		rPlungeCycleGrindFeedGeometry:=1.0;
		IF (iAutoProcess = 1) AND xMicroRodActive THEN
			rPlungeCycleGrindFeedGeometry:=T_AutoGeometryPara.rPlungeCycleGrindFeedGeometry;
		END_IF;
		T_WorkTool.rToolRotationSpeed:=rToolRotationSpeed;
		xCalculation:=TRUE;
		WHILE(xCalculation) DO
			(* calculate the grinding way of each section *)
			FBCalcPlungeGrindingMultiCycle(	T_Geometry:= T_Geometry,
											T_AutoGeometryPara:= T_AutoGeometryPara,
											rToolDiameter:= rToolDiameter,
											rToolDiameterWithOffset:=rToolDiameterWithOffset,
											rPlungeCycleGrindFeedGeometry:=rPlungeCycleGrindFeedGeometry,
											iStartSection:= iStartSection,
											iEndSection:= iEndSection,
											xReset:= xResetFB,
											xInit:=xInitFB);
			IF FBCalcPlungeGrindingMultiCycle.xEndWorking THEN		(* check if the end of the to work Tool is reached *)
				xCalculation:=FALSE;
				EXIT;
			END_IF;
			IF (FBCalcPlungeGrindingMultiCycle.iStepSectionWork = 7) THEN
				(* Count the Plunge Cycle *)
				T_WorkTool.iTotalCountDownPlungeCycle:=T_WorkTool.iTotalCountDownPlungeCycle + 1;
			END_IF;
			IF (FBCalcPlungeGrindingMultiCycle.iStepSectionWork >= 1) AND (FBCalcPlungeGrindingMultiCycle.iStepSectionWork <= 6) THEN
			(* section 1 - 6 *)
				iTmpStartSection:=iStartSection + (FBCalcPlungeGrindingMultiCycle.iStepSectionWork - 1);
				rGrindFeederPlunge:=FBCalcPlungeGrindingMultiCycle.rGrindingRelativePosition;
				T_WorkTool.rGrindFeederPlunge:=rGrindFeederPlunge;
				T_WorkTool.rPitch:=T_Geometry.arSectionPitch[iTmpStartSection];
				T_WorkTool.rToolLength:=T_Geometry.arSectionLength[iTmpStartSection];
				FBToolCalcul(	xMicroRodActive:=xMicroRodActive,
								xBeckhoffDriveActive:=FALSE,
								T_WorkTool:= T_WorkTool);
				rTimeLeftWork:=rTimeLeftWork + T_WorkTool.rTimeLeftWork;
			END_IF;
			IF (FBCalcPlungeGrindingMultiCycle.iStepSectionWork = 0) THEN
				(* Calc Plunge *)
				IF T_AutoGeometryPara.xPlungeActivationGeometry THEN
					T_WorkTool.rPitch:=T_Geometry.arSectionPitch[iStartSection] * -1.0;
					T_WorkTool.rGrindFeederPlunge:=FBCalcPlungeGrindingMultiCycle.rGrindingRelativePosition;
					rToolFeedLength:=T_AutoGeometryPara.rPlungeLengthToolFeedGeometry;
					T_WorkTool.rToolLength:=rToolFeedLength;
					T_WorkTool.rToolRotationSpeed:=T_AutoGeometryPara.rSpeedToolRotationGeometry;
					FBToolCalcul(	xMicroRodActive:=xMicroRodActive,
									xBeckhoffDriveActive:=FALSE,
									T_WorkTool:= T_WorkTool);
					rSpeedToolFeed:=T_WorkTool.rToolFeederSpeedUnit * -1.0;
					IF (rSpeedToolFeed <> 0) THEN
						rTimeLeftWork:=rTimeLeftWork + T_WorkTool.rToolLength/rSpeedToolFeed;
					END_IF;
				ELSE
					(* No Plunging activation, than also is the GrindFeeder the master *)
					rPlungeGrind:=ABS(FBCalcPlungeGrindingMultiCycle.rGrindingRelativePosition);
					IF (T_AutoGeometryPara.rPlungeSpeedGrindFeedGeometry <> 0) THEN
						rTimeLeftWork:=rTimeLeftWork + (rPlungeGrind / T_AutoGeometryPara.rPlungeSpeedGrindFeedGeometry);
					END_IF;
				END_IF;
			END_IF;
			IF (FBCalcPlungeGrindingMultiCycle.iStepSectionWork = 7) THEN
				(* Calc Displace *)
				IF T_AutoGeometryPara.xDisplaceActivationGeometry THEN
					T_WorkTool.rPitch:=T_Geometry.arSectionPitch[iEndSection] * -1.0;
					T_WorkTool.rGrindFeederPlunge:=FBCalcPlungeGrindingMultiCycle.rGrindingRelativePosition;
					rToolFeedLength:=T_AutoGeometryPara.rDisplaceLengthToolFeedGeometry;
					T_WorkTool.rToolLength:=rToolFeedLength;
					T_WorkTool.rToolRotationSpeed:=T_AutoGeometryPara.rSpeedToolRotationGeometry;
					FBToolCalcul(	xMicroRodActive:=xMicroRodActive,
									xBeckhoffDriveActive:=FALSE,
									T_WorkTool:= T_WorkTool);
					rSpeedToolFeed:=T_WorkTool.rToolFeederSpeedUnit * -1.0;
					IF (rSpeedToolFeed <> 0) THEN
						rTimeLeftWork:=rTimeLeftWork + T_WorkTool.rToolLength/rSpeedToolFeed;
					END_IF;
				ELSE
					(* No Displace activation, than also is the GrindFeeder the master *)
					rDisplaceGrind:=ABS(FBCalcPlungeGrindingMultiCycle.rGrindingRelativePosition);
					IF (T_AutoGeometryPara.rDisplaceSpeedGrindFeedGeometry <> 0) THEN
						rTimeLeftWork:=rTimeLeftWork + (rDisplaceGrind / T_AutoGeometryPara.rDisplaceSpeedGrindFeedGeometry);
					END_IF;
				END_IF;
			END_IF;
		END_WHILE;
		IF (T_AutoGeometryPara.iCycleGeometry > 1) THEN
			rTimeLeftWork:=rTimeLeftWork * INT_TO_REAL(T_AutoGeometryPara.iCycleGeometry);
		END_IF;
	END_IF;
(**************iAutoProcess 2 --> AutoGroove********************************************************************************************************************************************************************************************************)
	IF (iAutoProcess = 2) THEN
	(* calculate the time for the process AutoGeometry or AutoGroove *)
		T_WorkTool.iTotalCountDownPlungeCycle:=0;
		(* Check Start and End Section of the ToolGeometry *)
		FOR ii:=1 TO 6 DO
			IF T_Geometry.axActiveSection[ii] THEN
				IF (iStartSection = 0) THEN
					iStartSection:=ii;
				END_IF;
				iEndSection:=ii;
			END_IF;
		END_FOR;
(*
		xResetFB:=TRUE;
		(* reset first the FB for calculate the grinding plunge for each sections *)
		FBCalcPlungeGrinding(	rToolDiameter:= rToolDiameter,
								rToolDiameterWithOffset:=rToolDiameterWithOffset,
								xReset:= xResetFB);
		rPlungeCycleGrindFeedGeometry:=1.0;
*)
		xResetFB:=TRUE;
		(* reset first the FB for calculate the grinding plunge for each sections *)
		FBCalcPlungeGrindingMultiCycle(	rToolDiameter:= rToolDiameter,
										rToolDiameterWithOffset:=rToolDiameterWithOffset,
										xReset:= xResetFB,
										xInit:=xInitFB);
		xInitFB:=TRUE;
		FBCalcPlungeGrindingMultiCycle(	T_Geometry:= T_Geometry,
										T_AutoGeometryPara:= T_AutoGeometryPara,
										rToolDiameter:= rToolDiameter,
										rToolDiameterWithOffset:=rToolDiameterWithOffset,
										rPlungeCycleGrindFeedGeometry:=rPlungeCycleGrindFeedGeometry,
										iStartSection:= iStartSection,
										iEndSection:= iEndSection,
										xReset:= xResetFB,
										xInit:=xInitFB);
		rPlungeCycleGrindFeedGeometry:=1.0;
		IF (iAutoProcess = 2) OR NOT(xMicroRodActive) THEN
			rPlungeCycleGrindFeedGeometry:=rToolDiameter;		(* for the groove process or for the MicroWire is not possible to work in more cycle, because of that it will set the tooldiamter *)
		END_IF;
		T_WorkTool.rToolRotationSpeed:=rToolRotationSpeed;
		xCalculation:=TRUE;
		WHILE(xCalculation) DO
			(* calculate the grinding way of each section *)
			FBCalcPlungeGrindingMultiCycle(	T_Geometry:= T_Geometry,
											T_AutoGeometryPara:= T_AutoGeometryPara,
											rToolDiameter:= rToolDiameter,
											rToolDiameterWithOffset:=rToolDiameterWithOffset,
											rPlungeCycleGrindFeedGeometry:=rPlungeCycleGrindFeedGeometry,
											iStartSection:= iStartSection,
											iEndSection:= iEndSection,
											xReset:= xResetFB,
											xInit:=xInitFB);
			IF FBCalcPlungeGrindingMultiCycle.xEndWorking THEN		(* check if the end of the to work Tool is reached *)
				xCalculation:=FALSE;
				EXIT;
			END_IF;
			IF (T_WorkTool.iTotalCountDownPlungeCycle >= 20) THEN	(* not possible to work a Tool in more that 20 cycle *)
				xCalculation:=FALSE;
				EXIT;
			END_IF;
			IF (FBCalcPlungeGrindingMultiCycle.iStepSectionWork = 7) THEN
				(* Count the Plunge Cycle *)
				T_WorkTool.iTotalCountDownPlungeCycle:=T_WorkTool.iTotalCountDownPlungeCycle + 1;
			END_IF;
			IF (FBCalcPlungeGrindingMultiCycle.iStepSectionWork >= 1) AND (FBCalcPlungeGrindingMultiCycle.iStepSectionWork <= 6) THEN
			(* section 1 - 6 *)
				iTmpStartSection:=iStartSection + (FBCalcPlungeGrindingMultiCycle.iStepSectionWork - 1);
				rGrindFeederPlunge:=FBCalcPlungeGrindingMultiCycle.rGrindingRelativePosition;
				T_WorkTool.rGrindFeederPlunge:=rGrindFeederPlunge;
				T_WorkTool.rPitch:=T_AutoGroovePara.rPitchGroove;
				T_WorkTool.rToolLength:=T_Geometry.arSectionLength[iTmpStartSection];
				FBToolCalcul(	xMicroRodActive:=xMicroRodActive,
								xBeckhoffDriveActive:=FALSE,
								T_WorkTool:= T_WorkTool);
				rTimeLeftWork:=rTimeLeftWork + T_WorkTool.rTimeLeftWork;
			END_IF;
			IF (FBCalcPlungeGrindingMultiCycle.iStepSectionWork = 0) THEN
				(* Calc Plunge *)
				IF T_AutoGroovePara.xPlungeActivationGroove  THEN
					T_WorkTool.rPitch:=T_AutoGroovePara.rPitchGroove * -1.0;
					T_WorkTool.rGrindFeederPlunge:=FBCalcPlungeGrindingMultiCycle.rGrindingRelativePosition;
					rToolFeedLength:=T_AutoGroovePara.rPlungeLengthToolFeedGroove;
					T_WorkTool.rToolLength:=rToolFeedLength;
					T_WorkTool.rToolRotationSpeed:=T_AutoGroovePara.rSpeedToolRotationGroove;
					FBToolCalcul(	xMicroRodActive:=xMicroRodActive,
									xBeckhoffDriveActive:=FALSE,
									T_WorkTool:= T_WorkTool);
					rSpeedToolFeed:=T_WorkTool.rToolFeederSpeedUnit * -1.0;
					IF (rSpeedToolFeed <> 0) THEN
						rTimeLeftWork:=rTimeLeftWork + T_WorkTool.rToolLength/rSpeedToolFeed;
					END_IF;
				ELSE
					(* No Plunging activation, than also is the GrindFeeder the master *)
					rPlungeGrind:=ABS(FBCalcPlungeGrindingMultiCycle.rGrindingRelativePosition);
					IF (T_AutoGroovePara.rPlungeSpeedGrindFeedGroove <> 0) THEN
						rTimeLeftWork:=rTimeLeftWork + (rPlungeGrind / T_AutoGroovePara.rPlungeSpeedGrindFeedGroove);
					END_IF;
				END_IF;
			END_IF;
			IF (FBCalcPlungeGrindingMultiCycle.iStepSectionWork = 7) THEN
				(* Calc Displace *)
				IF T_AutoGroovePara.xDisplaceActivationGroove  THEN
					T_WorkTool.rPitch:=T_AutoGroovePara.rPitchGroove * -1.0;
					T_WorkTool.rGrindFeederPlunge:=FBCalcPlungeGrindingMultiCycle.rGrindingRelativePosition;
					rToolFeedLength:=T_AutoGroovePara.rDisplaceLengthToolFeedGroove;
					T_WorkTool.rToolLength:=rToolFeedLength;
					T_WorkTool.rToolRotationSpeed:=T_AutoGroovePara.rSpeedToolRotationGroove;
					FBToolCalcul(	xMicroRodActive:=xMicroRodActive,
									xBeckhoffDriveActive:=FALSE,
									T_WorkTool:= T_WorkTool);
					rSpeedToolFeed:=T_WorkTool.rToolFeederSpeedUnit * -1.0;
					IF (rSpeedToolFeed <> 0) THEN
						rTimeLeftWork:=rTimeLeftWork + T_WorkTool.rToolLength/rSpeedToolFeed;
					END_IF;
				ELSE
					(* No Displace activation, than also is the GrindFeeder the master *)
					rDisplaceGrind:=ABS(FBCalcPlungeGrindingMultiCycle.rGrindingRelativePosition);
					IF (T_AutoGroovePara.rDisplaceSpeedGrindFeedGroove <> 0) THEN
						rTimeLeftWork:=rTimeLeftWork + (rPlungeGrind / T_AutoGroovePara.rDisplaceSpeedGrindFeedGroove);
					END_IF;
				END_IF;
			END_IF;
		END_WHILE;
		IF (T_AutoGroovePara.iNumberOfGrooves > 1) THEN
			rTimeLeftWork:=rTimeLeftWork * INT_TO_REAL(T_AutoGroovePara.iNumberOfGrooves);
			(* Berechnung zusätzlicher Weg und Zeit für Ausstechen & Einstechen ab 2. Zyklus*)
			rPlungeGrind:=ABS(T_ProcessPara.rSecurityPosGrindFeedProcess - T_ProcessPara.rToolDiameterProcess) * 2.0;
			rTimeAddLeftWorkPlungeGrind:= rPlungeGrind / T_ProcessPara.rSpeedForwardFastGrindFeed;
			(* Berechnung zusätzlicher Weg und Zeit  Ausstechen für letzten Zyklus*)
			rPlungeGrind2:=ABS(T_ProcessPara.rSecurityPosGrindFeedProcess - T_ProcessPara.rToolDiameterProcess);
			rTimeAddLeftWorkPlungeGrind2:= rPlungeGrind2 / T_ProcessPara.rSpeedForwardFastGrindFeed;
			(*Berechnung zusätzlicher Weg und Zeit  Rückfahren  ab 2. Zyklus*)
			rToolLength:=0;
			FOR ii:=1 TO 6 DO
				IF T_Geometry.axActiveSection[ii] THEN
					rToolLength:=rToolLength + T_Geometry.arSectionLength[ii];
				END_IF;
			END_FOR;
			rTimeAddLeftWorkToolFeed:= rToolLength*10/T_ProcessPara.rSpeedStartPosToolFeedProcess;
			(*Berchnung der gesamten zusätzlichen Prozesszeit*)
			rTimeAddLeftWork:=(rTimeAddLeftWorkPlungeGrind + rTimeAddLeftWorkToolFeed) * (T_AutoGroovePara.iNumberOfGrooves -1);
			rTimeAddLeftWork:= rTimeAddLeftWork+rTimeAddLeftWorkPlungeGrind2;
			rTimeLeftWork:=rTimeLeftWork + rTimeAddLeftWork;
		END_IF;
	END_IF;
(**************iAutoProcess 0***********************************************************************************************************************************************************************************************************************)
	IF (iAutoProcess = 0) THEN
	(* Calculate the time for the process ToolCalibration *)
		T_WorkTool.rToolRotationSpeed:=T_CalibrationPara.rSpeedToolRotationCalib;
		T_WorkTool.rGrindFeederPlunge:=T_ProcessPara.rOffsetBeforeToolDiaGrindFeedProcess;
		T_WorkTool.rPitch:=T_CalibrationPara.rPitchCalib;
		T_WorkTool.rToolLength:=T_CalibrationPara.rToolLengthCylinderPartCalib;
		FBToolCalcul(	xMicroRodActive:=xMicroRodActive,
						xBeckhoffDriveActive:=FALSE,
						T_WorkTool:= T_WorkTool);
		rTimeLeftWork:=rTimeLeftWork + T_WorkTool.rTimeLeftWork;
		IF T_CalibrationPara.xPlungeActivationCalib THEN
			T_WorkTool.rPitch:=T_CalibrationPara.rPitchCalib;
			T_WorkTool.rGrindFeederPlunge:=T_ProcessPara.rOffsetBeforeToolDiaGrindFeedProcess;
			rToolFeedLength:=T_CalibrationPara.rPlungeLengthToolFeedCalib;
			T_WorkTool.rToolLength:=rToolFeedLength;
			FBToolCalcul(	xMicroRodActive:=xMicroRodActive,
							xBeckhoffDriveActive:=FALSE,
							T_WorkTool:= T_WorkTool);
			rSpeedToolFeed:=T_WorkTool.rToolFeederSpeedUnit;
			IF (rSpeedToolFeed <> 0) THEN
				rTimeLeftWork:=rTimeLeftWork + T_WorkTool.rToolLength/ABS(rSpeedToolFeed);
			END_IF;
		ELSE
			(* No Plunging activation, than also is the GrindFeeder the master *)
			rPlungeGrind:=T_ProcessPara.rOffsetBeforeToolDiaGrindFeedProcess;
			rTimeLeftWork:=rTimeLeftWork + (rPlungeGrind / T_CalibrationPara.rPlungeSpeedGrindFeedCalib);
		END_IF;


		IF T_CalibrationPara.xDisplaceActivationCalib THEN
			T_WorkTool.rPitch:=T_CalibrationPara.rPitchCalib * -1.0;
			T_WorkTool.rGrindFeederPlunge:=T_ProcessPara.rOffsetBeforeToolDiaGrindFeedProcess;
			rToolFeedLength:=T_CalibrationPara.rDisplaceLengthToolFeedCalib;
			T_WorkTool.rToolLength:=rToolFeedLength;
			FBToolCalcul(	xMicroRodActive:=xMicroRodActive,
							xBeckhoffDriveActive:=FALSE,
							T_WorkTool:= T_WorkTool);
			rSpeedToolFeed:=T_WorkTool.rToolFeederSpeedUnit;
			IF (rSpeedToolFeed <> 0) THEN
				rTimeLeftWork:=rTimeLeftWork + T_WorkTool.rToolLength/ABS(rSpeedToolFeed);
			END_IF;
		ELSE
			(* No Displace activation, than also is the GrindFeeder the master *)
			rDisplaceGrind:=T_ProcessPara.rOffsetBeforeToolDiaGrindFeedProcess;
			rTimeLeftWork:=rTimeLeftWork + (rDisplaceGrind / T_CalibrationPara.rDisplaceSpeedGrindFeedCalib);
		END_IF;
	END_IF;
	rProcessTime:=rTimeLeftWork;
END_FUNCTION_BLOCK

(* POU GENERAL/FB_TOOL_CALCUL, ST *)
FUNCTION_BLOCK FB_TOOL_CALCUL
VAR_INPUT
	xMicroRodActive: BOOL;			(* choice of the machine MicroWire or MicroRod *)
	xBeckhoffDriveActive: BOOL;		(* choice of the Axis Beckhoff or EcoStep *)
END_VAR
VAR_IN_OUT
	T_WorkTool:ST_WORKTOOL;		(* Tool Parameter *)
END_VAR
VAR_OUTPUT
END_VAR
VAR
END_VAR
(****************************************************************************************************************************************************)
(***********                                  This Functionblock calculate all needed parameter for work a Tool                                            ************)
(****************************************************************************************************************************************************)
(* calcul ToolRotation Speed in inc/64s *)
	IF (T_WorkTool.rToolRotationSpeed <> 0) AND (T_WorkTool.rToolRightGearRatio <> 0) THEN
		T_WorkTool.rToolRotationSpeedMotor:=((T_WorkTool.rToolRotationSpeed / 60.0) * 8000.0 * 64.0) / T_WorkTool.rToolRightGearRatio;
	ELSE
		RETURN;	(* Exit FB *)
	END_IF;
(* calcul ToolFeeder Speed in mm/s *)
	T_WorkTool.rToolFeederSpeedUnit:=T_WorkTool.rPitch * (T_WorkTool.rToolRotationSpeed / 60.0);
(* calcul ToolFeeder Speed in inc/64s Relativ *)
	T_WorkTool.rToolFeederSpeedMotorRel:=T_WorkTool.rToolFeederScaleFactor * T_WorkTool.rToolFeederSpeedUnit * 64.0;
(* calcul ToolFeeder Speed in inc/64s Relativ *)
	T_WorkTool.rToolFeederSpeedMotorAbs:=(T_WorkTool.rToolRotationSpeedMotor * T_WorkTool.rToolRightGearRatio) + T_WorkTool.rToolFeederSpeedMotorRel;
(* Set ToolFeeder GearDivider *)
	T_WorkTool.iToolFeederGearDivider:=T_WorkTool.iBaseGearDivider;
	IF xMicroRodActive THEN
	(* calcul ToolFeeder GearFactor *)
		IF (T_WorkTool.rPitch <> 0) THEN
			T_WorkTool.iToolFeederGearFactor:=REAL_TO_INT(INT_TO_REAL(T_WorkTool.iBaseGearDivider) / (T_WorkTool.rToolRotationSpeedMotor / T_WorkTool.rToolFeederSpeedMotorRel));
		ELSE
			T_WorkTool.iToolFeederGearFactor:=REAL_TO_INT(INT_TO_REAL(T_WorkTool.iToolFeederGearDivider) * T_WorkTool.rToolRightGearRatio);
		END_IF;
	ELSE
	(* calcul ToolFeeder GearFactor *)
		IF (T_WorkTool.rPitch <> 0) THEN
			T_WorkTool.iToolFeederGearFactor:=REAL_TO_INT(INT_TO_REAL(T_WorkTool.iBaseGearDivider) / (T_WorkTool.rToolRotationSpeedMotor / T_WorkTool.rToolFeederSpeedMotorAbs));
		ELSE
			T_WorkTool.iToolFeederGearFactor:=REAL_TO_INT(INT_TO_REAL(T_WorkTool.iToolFeederGearDivider) * T_WorkTool.rToolRightGearRatio);
		END_IF;
	END_IF;
(* calcul Time to work *)
	IF (T_WorkTool.rToolFeederSpeedUnit <> 0) THEN
		T_WorkTool.rTimeLeftWork:=(T_WorkTool.rToolLength * 10.0) / ABS(T_WorkTool.rToolFeederSpeedUnit);
	ELSE
		T_WorkTool.rTimeLeftWork:=0.0;
	END_IF;
(* calcul ToolFeeder relative Position to drive *)
	T_WorkTool.rToolFeederRelPositionUnit:=T_WorkTool.rToolLength * 10.0;
	T_WorkTool.rToolFeederRelPositionMotor:=T_WorkTool.rToolFeederRelPositionUnit * T_WorkTool.rToolFeederScaleFactor;
(* calcul GrindFeeder Speed in um/s *)
	IF (T_WorkTool.rTimeLeftWork <> 0) THEN
		T_WorkTool.rGrindFeederSpeedUnit:=T_WorkTool.rGrindFeederPlunge / T_WorkTool.rTimeLeftWork;
	ELSE
		T_WorkTool.rGrindFeederSpeedUnit:=0.0;
	END_IF;
(* calcul GrindFeeder Speed in inc/s *)
	T_WorkTool.rGrindFeederSpeedMotor:=T_WorkTool.rGrindFeederSpeedUnit * T_WorkTool.rGrindFeederScaleFactor * 64.0;
END_FUNCTION_BLOCK

(* POU GENERAL/FB_CALC_PLUNGE_GRINDING, ST *)
FUNCTION_BLOCK FB_CALC_PLUNGE_GRINDING
VAR_INPUT
	T_Geometry:ST_GEOMETRY;								(* Structure of the NovRAM parameter *)
	T_AutoGeometryPara:ST_EXCHG_PARAM_AUTOGEOMETRY;	(* Structure of the NovRAM parameter *)
	rToolDiameter:REAL;					(* diameter of the unworked Tool *)
	rToolDiameterWithOffset:REAL;			(* diameter of the unworked Tool plus the offset for plunge and displace procedure *)
	rPlungeCycleGrindFeedGeometry:REAL;	(* max grinding plunging per cycle *)
	iStartSection:INT;						(* number of the start section *)
	iEndSection:INT;						(* number of the end section *)
END_VAR
VAR_IN_OUT
	xReset:BOOL;						(* resetting of the FB *)
END_VAR
VAR_OUTPUT
	iStepSectionWork:INT;				(* actual worked section number *)
	rGrindingRelativePosition:REAL;		(* relative way of the GrindFeeder plunge *)
	xEndWorking:BOOL;				(* end of the hole working procedure *)
	xError:BOOL;						(* error flag *)
END_VAR
VAR
(***S***)
	rActualPositionGrindFeedStart: ARRAY [0..7] OF REAL;	(* 0=StartPos Plunge,1-6=Dynamic StartPos Section 1-6, 7=StartPos Displace *)
	rActualPositionGrindFeedEnd: ARRAY [0..7] OF REAL;	(* 0=EndPos Plunge,1-6=Dynamic EndPos Section 1-6, 7=EndPos Displace *)
	rDistanceToWorkedTool: REAL;
	ii: INT;
	iStepSection: INT;
	axWorkEndSection: ARRAY [0..7] OF BOOL;
	xCheckEnd: BOOL;
	rTmpActualPositionGrindFeedStart:REAL;
	iStepCheckSection: INT;
	rTmpDistance: REAL;
	rGrinded: REAL;
END_VAR
(****************************************************************************************************************************************************)
(***********      This Functionblock calculate the plunge way for the GrindFeeder axis for the geometry sections  1-6        ************)
(***********                                           It calculate also the plunge and displace procedure							    ************)
(****************************************************************************************************************************************************)
IF xReset THEN
	xReset:=FALSE;
	iStepSection:=0;
	FOR ii:=0 TO 7 DO
		rActualPositionGrindFeedStart[ii]:=rToolDiameterWithOffset;
		rActualPositionGrindFeedEnd[ii]:=rToolDiameterWithOffset;
		axWorkEndSection[ii]:=FALSE;
	END_FOR;
	rActualPositionGrindFeedStart[0]:=rToolDiameterWithOffset;
	rActualPositionGrindFeedEnd[7]:=rToolDiameterWithOffset;
	rTmpActualPositionGrindFeedStart:=rToolDiameterWithOffset;
	rGrindingRelativePosition:=0.0;
	iStepSectionWork:=0;
	RETURN;
END_IF;
xError:=FALSE;
(* check the settled start and end section *)
IF (iStartSection < 1) OR (iStartSection > 6) THEN
	xError:=TRUE;
	RETURN;
END_IF;
IF (iEndSection < 1) OR (iEndSection > 6) THEN
	xError:=TRUE;
	RETURN;
END_IF;
IF (iStepSection < 0) OR (iStepSection > 7) THEN
	xError:=TRUE;
	RETURN;
END_IF;

CASE iStepSection OF
	(* plunge procedure *)
		0:	iStepCheckSection:=1;
			xCheckEnd:=TRUE;
			(* Check if the end of all section is reached *)
			FOR ii:=iStartSection TO iEndSection DO
				IF (rActualPositionGrindFeedStart[iStepCheckSection] <> T_Geometry.arStartDiameter[ii]) THEN
					xCheckEnd:=FALSE;
				END_IF;
				IF (rActualPositionGrindFeedEnd[iStepCheckSection] <> T_Geometry.arEndDiameter[ii]) THEN
					xCheckEnd:=FALSE;
				END_IF;
				iStepCheckSection:=iStepCheckSection + 1;
			END_FOR;
			xEndWorking:=xCheckEnd;
			IF xEndWorking THEN
				rGrindingRelativePosition:=0.0;
				RETURN;
			END_IF;
			IF (T_Geometry.arStartDiameter[iStartSection] = rActualPositionGrindFeedEnd[0]) THEN	(* check if the defined ToolDiameter for the plunge procedure is reached *)
				axWorkEndSection[0]:=TRUE;
				rGrindingRelativePosition:=rToolDiameterWithOffset - T_Geometry.arStartDiameter[iStartSection];
			END_IF;
			IF NOT(axWorkEndSection[0]) THEN
			(* if the end of the plunge procedure is not reached, then calculate the plunge way of the plunge procedure *)
				rGrindingRelativePosition:=(rToolDiameterWithOffset - rActualPositionGrindFeedEnd[0]) + rPlungeCycleGrindFeedGeometry;
				IF ((rToolDiameterWithOffset - rGrindingRelativePosition) <= T_Geometry.arStartDiameter[iStartSection]) THEN
					rGrindingRelativePosition:=rToolDiameterWithOffset - T_Geometry.arStartDiameter[iStartSection];
				END_IF;
			END_IF;
			rActualPositionGrindFeedStart[0]:=rToolDiameterWithOffset;	(* the start zero section of the geometry is always the diameter of the Tool *)
			rActualPositionGrindFeedEnd[0]:=rToolDiameterWithOffset - rGrindingRelativePosition;	(* calcualte the plunge way *)
			iStepSectionWork:=iStepSection;	(* set the actual section which is working *)
			iStepSection:=iStepSection + 1;		(* go to the next section *)
	(* geometry section 1,2,3,4,5 and 6 *)
	1,2,3,4,5,6:	rGrinded:=(rActualPositionGrindFeedStart[iStepSection] - rActualPositionGrindFeedEnd[iStepSection - 1]);	(* calculate the difference of the worked section before to the unworked section after *)
			IF (rGrinded < 0) THEN
				rGrinded:=rGrinded;
			END_IF;
			rActualPositionGrindFeedStart[iStepSection]:=rActualPositionGrindFeedStart[iStepSection] - rGrinded;		(* set the new diameter of the section which will go to work *)
			rTmpDistance:=T_Geometry.arStartDiameter[iStartSection + (iStepSection - 1)] - T_Geometry.arEndDiameter[iStartSection + (iStepSection - 1)]; (* set the difference of the start and end diameter of the section *)
			IF (rActualPositionGrindFeedStart[iStepSection] < T_Geometry.arStartDiameter[iStartSection + (iStepSection - 1)]) THEN	(* correct of the to grind Tool diameter *)
				rActualPositionGrindFeedStart[iStepSection]:=T_Geometry.arStartDiameter[iStartSection + (iStepSection - 1)];
			END_IF;
			rGrindingRelativePosition:=rPlungeCycleGrindFeedGeometry - rGrinded;	(* calculate the effectiv way for the plunge *)
			IF (rGrinded >= rPlungeCycleGrindFeedGeometry) THEN				(* check if the to grinding way is grater than the defined max grinding *)
				IF (rActualPositionGrindFeedStart[iStepSection] < T_Geometry.arEndDiameter[iStartSection + (iStepSection - 1)]) THEN
				(* correct the effective way for the plunge, because it can not work more than the defined grinding way *)
					rGrindingRelativePosition:=rActualPositionGrindFeedStart[iStepSection] - T_Geometry.arEndDiameter[iStartSection + (iStepSection - 1)];
				END_IF;
			ELSE
				IF (rTmpDistance = 0) THEN
				(* a cylinder part will now work *)
					rGrindingRelativePosition:=0.0;
				ELSE
					(* a cone part will now work *)
					rTmpDistance:=T_Geometry.arStartDiameter[iStartSection + (iStepSection - 1)] - rActualPositionGrindFeedEnd[iStepSection];
					rGrindingRelativePosition:=rTmpDistance + rPlungeCycleGrindFeedGeometry;
					IF ((T_Geometry.arStartDiameter[iStartSection + (iStepSection - 1)] - rGrindingRelativePosition) < T_Geometry.arEndDiameter[iStartSection + (iStepSection - 1)]) THEN
					(* correct the effective way for the plunge, because it can not work more than the defined grinding way *)
						rGrindingRelativePosition:=T_Geometry.arStartDiameter[iStartSection + (iStepSection - 1)] - T_Geometry.arEndDiameter[iStartSection + (iStepSection - 1)];
					END_IF;
				END_IF;
			END_IF;
			rActualPositionGrindFeedEnd[iStepSection]:=rActualPositionGrindFeedStart[iStepSection] - rGrindingRelativePosition;	(* calculate the end position of the section *)
			iStepSectionWork:=iStepSection;		(* set the actual section which is working *)
			IF ((iStepSection + (iStartSection - 1)) < iEndSection) THEN	(* check if the end section is active *)
				iStepSection:=iStepSection + 1;
			ELSE
				iStepSection:=7;	(* end section is reached-->go the displace procedure *)
			END_IF;
	(* plunge procedure *)
	7:		rActualPositionGrindFeedStart[7]:=rActualPositionGrindFeedEnd[iEndSection - (iStartSection - 1)];	(* set the new diameter of the section which will going to work *)
			rDistanceToWorkedTool:=rActualPositionGrindFeedStart[7] - rToolDiameterWithOffset;	(* check the distance to the end diameter, which will go to work *)
			rGrindingRelativePosition:=rDistanceToWorkedTool;
			IF (rActualPositionGrindFeedStart[5] = T_Geometry.arEndDiameter[iEndSection]) THEN
				axWorkEndSection[7]:=TRUE;		(* the end of this section is reached *)
			ELSE
				axWorkEndSection[7]:=FALSE;		(* the end of this section is reached *)
			END_IF;
			rActualPositionGrindFeedEnd[7]:=rToolDiameterWithOffset;
			iStepSectionWork:=iStepSection;		(* set the actual section which is working *)
			iStepSection:=0;
END_CASE;
END_FUNCTION_BLOCK

(* POU GENERAL/FB_CALC_PLUNGE_GRINDING_MultiCycle, ST *)
FUNCTION_BLOCK FB_CALC_PLUNGE_GRINDING_MultiCycle
VAR_INPUT
	T_Geometry:ST_GEOMETRY;								(* Structure of the NovRAM parameter *)
	T_AutoGeometryPara:ST_EXCHG_PARAM_AUTOGEOMETRY;	(* Structure of the NovRAM parameter *)
	rToolDiameter:REAL;					(* diameter of the unworked Tool *)
	rToolDiameterWithOffset:REAL;			(* diameter of the unworked Tool plus the offset for plunge and displace procedure *)
	rPlungeCycleGrindFeedGeometry:REAL;	(* max grinding plunging per cycle *)
	iStartSection:INT;						(* number of the start section *)
	iEndSection:INT;						(* number of the end section *)
END_VAR
VAR_IN_OUT
	xReset:BOOL;						(* resetting of the FB *)
	xInit:BOOL;							(* Init of the FB *)
END_VAR
VAR_OUTPUT
	iStepSectionWork:INT;				(* actual worked section number *)
	rGrindingRelativePosition:REAL;		(* relative way of the GrindFeeder plunge *)
	xEndWorking:BOOL;				(* end of the hole working procedure *)
	xError:BOOL;						(* error flag *)
END_VAR
VAR
	rActualPositionGrindFeedStart: ARRAY [0..7] OF REAL;	(* 0=StartPos Plunge,1-4=Dynamic StartPos Section 1-4, 5=StartPos Displace *)
	rActualPositionGrindFeedEnd: ARRAY [0..7] OF REAL;	(* 0=EndPos Plunge,1-4=Dynamic EndPos Section 1-4, 5=EndPos Displace *)
	rDistanceToWorkedTool: REAL;
	ii: INT;
	iStepSection: INT;
	axWorkEndSection: ARRAY [0..7] OF BOOL;
	xCheckEnd: BOOL;
	rTmpActualPositionGrindFeedStart:REAL;
	iStepCheckSection: INT;
	rTmpDistance: REAL;
	rGrinded: REAL;
	rMaxPlungeWay:REAL;
	rMaxPlungeWayStepOffset:REAL;
        	diNrOfAdditionalPlungeCycle:DINT;
END_VAR
(*****************************************************************************************************************************************************)
(***********      This Functionblock calculates the plunge way for the GrindFeeder axis for the geometry sections  1-6        ************)
(***********                                           It calculates also the plunge and displace procedure							    *************)
(*****************************************************************************************************************************************************)
IF xReset THEN
	xReset:=FALSE;
	iStepSection:=0;
	FOR ii:=0 TO 7 DO
		rActualPositionGrindFeedStart[ii]:=rToolDiameterWithOffset;
		rActualPositionGrindFeedEnd[ii]:=rToolDiameterWithOffset;
		axWorkEndSection[ii]:=FALSE;
	END_FOR;
	rActualPositionGrindFeedStart[0]:=rToolDiameterWithOffset;
	rActualPositionGrindFeedEnd[7]:=rToolDiameterWithOffset;
	rTmpActualPositionGrindFeedStart:=rToolDiameterWithOffset;
	rGrindingRelativePosition:=0.0;
	iStepSectionWork:=0;
	rMaxPlungeWay:=0.0;
	RETURN;
END_IF;
(*22.12.2009: KFS 	{   *)
IF xInit THEN
	xInit:=FALSE;
(*	rMaxPlungeWay:= rToolDiameter - T_Geometry.arEndDiameter[iEndSection]; (*Calculation of the max. plunge way*)*)
	rMaxPlungeWay:= rToolDiameterWithOffset - T_Geometry.arEndDiameter[iEndSection]; (*Calculation of the max. plunge way*)
	diNrOfAdditionalPlungeCycle:= MODTURNS (rMaxPlungeWay, rPlungeCycleGrindFeedGeometry);
	IF diNrOfAdditionalPlungeCycle > 0 THEN
		rMaxPlungeWayStepOffset:=LMOD(rMaxPlungeWay, rPlungeCycleGrindFeedGeometry);
		IF rMaxPlungeWayStepOffset > 0 THEN
			diNrOfAdditionalPlungeCycle:=diNrOfAdditionalPlungeCycle + 1;
		END_IF;
		rMaxPlungeWay:= rPlungeCycleGrindFeedGeometry * diNrOfAdditionalPlungeCycle;
	END_IF;
	iStepCheckSection:=1;
	(*Add the max plunge way on all start- and stop- points of the geometry*)
	FOR ii:=iStartSection TO iEndSection DO
(*		rActualPositionGrindFeedStart[iStepCheckSection] := rToolDiameterWithOffset - rToolDiameter +T_Geometry.arStartDiameter[ii] + rMaxPlungeWay;
		rActualPositionGrindFeedEnd[iStepCheckSection]:= rToolDiameterWithOffset  - rToolDiameter + T_Geometry.arEndDiameter[ii]+ rMaxPlungeWay; *)
		rActualPositionGrindFeedStart[iStepCheckSection] := T_Geometry.arStartDiameter[ii] + rMaxPlungeWay;
		rActualPositionGrindFeedEnd[iStepCheckSection]:=  T_Geometry.arEndDiameter[ii]+ rMaxPlungeWay;
		iStepCheckSection:=iStepCheckSection + 1;
	END_FOR;
	rActualPositionGrindFeedStart[0]:=rActualPositionGrindFeedStart[1];
	rActualPositionGrindFeedEnd[0]:=rActualPositionGrindFeedStart[1];
	RETURN;
END_IF;
(*22.12.2009: KFS 	}   *)
xError:=FALSE;
(* check the settled start and end section *)
IF (iStartSection < 1) OR (iStartSection > 6) THEN
	xError:=TRUE;
	RETURN;
END_IF;
IF (iEndSection < 1) OR (iEndSection > 6) THEN
	xError:=TRUE;
	RETURN;
END_IF;
IF (iStepSection < 0) OR (iStepSection > 7) THEN
	xError:=TRUE;
	RETURN;
END_IF;
CASE iStepSection OF
	(* plunge procedure *)
		0:	iStepCheckSection:=1;
			xCheckEnd:=TRUE;
			(* Check if the end of all section is reached *)
			FOR ii:=iStartSection TO iEndSection DO
				IF (rActualPositionGrindFeedStart[iStepCheckSection] <> T_Geometry.arStartDiameter[ii]) THEN
					xCheckEnd:=FALSE;
				END_IF;
				IF (rActualPositionGrindFeedEnd[iStepCheckSection] <> T_Geometry.arEndDiameter[ii]) THEN
					xCheckEnd:=FALSE;
				END_IF;
				iStepCheckSection:=iStepCheckSection + 1;
			END_FOR;
			xEndWorking:=xCheckEnd;
			IF xEndWorking THEN
				rGrindingRelativePosition:=0.0;
				RETURN;
			END_IF;
			IF (T_Geometry.arStartDiameter[iStartSection] = rActualPositionGrindFeedEnd[0]) THEN	(* check if the defined ToolDiameter for the plunge procedure is reached *)
				axWorkEndSection[0]:=TRUE;
				rGrindingRelativePosition:=rToolDiameterWithOffset - T_Geometry.arStartDiameter[iStartSection];
			END_IF;
			IF NOT(axWorkEndSection[0]) THEN
			(* if the end of the plunge procedure is not reached, then calculate the plunge way of the plunge procedure *)
				rGrindingRelativePosition:=(rToolDiameterWithOffset - rActualPositionGrindFeedEnd[0]) + rPlungeCycleGrindFeedGeometry;
				IF ((rToolDiameterWithOffset - rGrindingRelativePosition) <= T_Geometry.arStartDiameter[iStartSection]) THEN
					rGrindingRelativePosition:=rToolDiameterWithOffset - T_Geometry.arStartDiameter[iStartSection];
				END_IF;
			END_IF;
			(*22.12.2009: KFS 	{   *)
			(*
			rActualPositionGrindFeedStart[0]:=rToolDiameterWithOffset;	(* the start zero section of the geometry is always the diameter of the Tool *)
			*)
			rActualPositionGrindFeedStart[0]:=rToolDiameterWithOffset - rGrindingRelativePosition;	(* the start zero section of the geometry is always the diameter of the Tool *)
			(*22.12.2009: KFS 	}   *)
			rActualPositionGrindFeedEnd[0]:=rToolDiameterWithOffset - rGrindingRelativePosition;	(* calcualte the plunge way *)
			iStepSectionWork:=iStepSection;	(* set the actual section which is working *)
			iStepSection:=iStepSection + 1;		(* go to the next section *)
	(* geometry section 1,2,3, 4,5 and 6 *)
	1..6:	rGrinded:=(rActualPositionGrindFeedStart[iStepSection] - rActualPositionGrindFeedEnd[iStepSection - 1]);	(* calculate the difference of the worked section before to the unworked section after *)
			IF (rGrinded < 0) THEN
				rGrinded:=rGrinded;
			END_IF;
			rActualPositionGrindFeedStart[iStepSection]:=rActualPositionGrindFeedStart[iStepSection] - rGrinded;		(* set the new diameter of the section which will going to work *)
			rTmpDistance:=T_Geometry.arStartDiameter[iStartSection + (iStepSection - 1)] - T_Geometry.arEndDiameter[iStartSection + (iStepSection - 1)]; (* set the difference of the start and end diameter of the section *)
			IF (rActualPositionGrindFeedStart[iStepSection] < T_Geometry.arStartDiameter[iStartSection + (iStepSection - 1)]) THEN	(* correct of the to grind Tool diameter *)
				rActualPositionGrindFeedStart[iStepSection]:=T_Geometry.arStartDiameter[iStartSection + (iStepSection - 1)];
			END_IF;
			rGrindingRelativePosition:=rPlungeCycleGrindFeedGeometry - rGrinded ;	(* calculate the effectiv way for the plunge *)
(*			IF (rGrinded >= rPlungeCycleGrindFeedGeometry) THEN				(* check if the to grinding way is grater than the defined max grinding *) *)
			IF (rGrinded > rPlungeCycleGrindFeedGeometry) THEN				(* check if the to grinding way is grater than the defined max grinding *)
				IF (rActualPositionGrindFeedStart[iStepSection] < T_Geometry.arEndDiameter[iStartSection + (iStepSection - 1)]) THEN
				(* correct the effective way for the plunge, because it can not work more than the defined grinding way *)
					rGrindingRelativePosition:=rActualPositionGrindFeedStart[iStepSection] - T_Geometry.arEndDiameter[iStartSection + (iStepSection - 1)];
				END_IF;
			ELSE
				IF (rTmpDistance = 0) THEN
				(* a cylinder part will now work *)
					rGrindingRelativePosition:=0.0;
				ELSE
					(* a cone part will now work *)
					rGrindingRelativePosition:=rTmpDistance;
					IF ((T_Geometry.arStartDiameter[iStartSection + (iStepSection - 1)] - rGrindingRelativePosition) < T_Geometry.arEndDiameter[iStartSection + (iStepSection - 1)]) THEN
					(* correct the effective way for the plunge, because it can not work more than the defined grinding way *)
						rGrindingRelativePosition:=T_Geometry.arStartDiameter[iStartSection + (iStepSection - 1)] - T_Geometry.arEndDiameter[iStartSection + (iStepSection - 1)];
					END_IF;
				END_IF;
			END_IF;
			rActualPositionGrindFeedEnd[iStepSection]:=rActualPositionGrindFeedStart[iStepSection] - rGrindingRelativePosition;	(* calculate the end position of the section *)

			iStepSectionWork:=iStepSection;		(* set the actual section which is working *)
			IF ((iStepSection + (iStartSection - 1)) < iEndSection) THEN	(* check if the end section is active *)
				iStepSection:=iStepSection + 1;
			ELSE
				iStepSection:=7;	(* end section is reached-->go the displace procedure *)
			END_IF;
	(* plunge procedure *)
	7:		rActualPositionGrindFeedStart[7]:=rActualPositionGrindFeedEnd[iEndSection - (iStartSection - 1)];	(* set the new diameter of the section which will going to work *)
			rDistanceToWorkedTool:=rActualPositionGrindFeedStart[7] - rToolDiameterWithOffset;	(* check the distance to the end diameter, which will go to work *)
			rGrindingRelativePosition:=rDistanceToWorkedTool;
			IF (rActualPositionGrindFeedStart[7] = T_Geometry.arEndDiameter[iEndSection]) THEN
				axWorkEndSection[7]:=TRUE;		(* the end of this section is reached *)
			ELSE
				axWorkEndSection[7]:=FALSE;		(* the end of this section is not reached *)
			END_IF;
			rActualPositionGrindFeedEnd[7]:=rToolDiameterWithOffset;
			iStepSectionWork:=iStepSection;		(* set the actual section which is working *)
			iStepSection:=0;
END_CASE;
END_FUNCTION_BLOCK

(* POU PRG_VISU_LAYER5/FB_VISU/iFctGetEditParaList, ST *)
FUNCTION iFctGetEditParaList : INT
VAR_INPUT
	dwActualPage:DWORD;		(* activate page on the visualisation *)
	xMicroRodActive: BOOL;		(* choice of the machine MicroWire or MicroRod *)
	iSelectParaList:INT;			(* parameter list choiced on the QVis *)
	iSelectParaListTeachRot:INT;	(* parameter list choiced on the QVis for teach ToolRotation *)
END_VAR
VAR
	iTmpRetEditParaList: INT;
END_VAR
(****************************************************************************************************************************************************)
(***********          This Function check the state of the parameter level and give the number of the parameter list                ************)
(****************************************************************************************************************************************************)
iTmpRetEditParaList:=0;
CASE dwActualPage OF
	110:	IF xMicroRodActive THEN
			iTmpRetEditParaList:=111;
		ELSE
			iTmpRetEditParaList:=110;
		END_IF;
	120:	IF (iSelectParaList = 0) OR (iSelectParaList = 1) THEN
			IF xMicroRodActive THEN
				iTmpRetEditParaList:=123;
			ELSE
				iTmpRetEditParaList:=120;
			END_IF;
		END_IF;
		IF (iSelectParaList = 2) THEN
			iTmpRetEditParaList:=121;
		END_IF;
		IF (iSelectParaList = 3) THEN
			IF xMicroRodActive THEN
				iTmpRetEditParaList:=125;
			ELSE
				iTmpRetEditParaList:=122;
			END_IF;
		END_IF;
	130:	IF xMicroRodActive THEN
			iTmpRetEditParaList:=131;
		ELSE
			iTmpRetEditParaList:=130;
		END_IF;
	140:	iTmpRetEditParaList:=140;
	150:	iTmpRetEditParaList:=150;
	210:	IF (iSelectParaListTeachRot = 0) OR (iSelectParaListTeachRot = 1) THEN
			iTmpRetEditParaList:=210;
		END_IF;
		IF (iSelectParaListTeachRot = 2) THEN
			iTmpRetEditParaList:=211;
		END_IF;
		IF (iSelectParaListTeachRot = 3) THEN
			iTmpRetEditParaList:=212;
		END_IF;
	220:	iTmpRetEditParaList:=0;
	230:	iTmpRetEditParaList:=230;
	310:IF xMicroRodActive THEN
			iTmpRetEditParaList:=311;
		ELSE
			iTmpRetEditParaList:=310;
		END_IF;
	320:	iTmpRetEditParaList:=0;
	410:	iTmpRetEditParaList:=410;
	420:	iTmpRetEditParaList:=0;
	430:	iTmpRetEditParaList:=0;
END_CASE;
iFctGetEditParaList:=iTmpRetEditParaList;
END_FUNCTION

(* POU PRG_VISU_LAYER5/FB_VISU/iFctReturnConfMessage, ST *)
FUNCTION iFctReturnConfMessage : INT
VAR_INPUT
	iNumAction:INT;	(* number of called action on the visualisation *)
END_VAR
VAR
END_VAR
(****************************************************************************************************************************************************)
(***********                      This Function check the action on the visu and gives a correspond message number                     ************)
(****************************************************************************************************************************************************)
	CASE iNumAction OF
	(* Action exceeded Timeout *)
	-1:	iFctReturnConfMessage:=102;
	(* NovRAM, 'Parameter saved' with confirmation *)
	1005:	iFctReturnConfMessage:=1;
	(* NovRAM, 'Parameter saved' without confirmation *)
	1006:	iFctReturnConfMessage:=1;
	(* Reference machine done *)
	1110:	iFctReturnConfMessage:=23;
	(* Process machine done *)
	1150:	iFctReturnConfMessage:=21;
	(* Process station done *)
	1151..1153:	iFctReturnConfMessage:=22;
	(* change page, no message *)
	10001..10999:	iFctReturnConfMessage:=0;
	(* Info , 'Confirm action' *)
	ELSE	iFctReturnConfMessage:=2;
	END_CASE
END_FUNCTION

(* POU PRG_VISU_LAYER5/FB_VISU/xFctCtrleProfileName, ST *)
FUNCTION xFctCtrleProfileName : BOOL
VAR_INPUT
	sNewProfileName:STRING(30);		(* profile name to save *)
	ptrProfileList:POINTER TO ARRAY[1..csiMaxProfile] OF ST_PROFILE_ID;	(* list of the saved profil names *)
END_VAR
VAR
(* variable *)
	i: INT;
	sTmp:STRING;
	sTmp2:STRING;
END_VAR
(****************************************************************************************************************************************************)
(***********                                              This Function check the name of the profile if it is correct                                                     ************)
(****************************************************************************************************************************************************)
(* Init. function *)
	xFctCtrleProfileName:=FALSE;
	sTmp:=FCT_UPLOW_CASE(	xLowConvert:=TRUE,
							sInString:=sNewProfileName);

(* Search if name already exists *)
	FOR i:=1 TO csiMaxProfile DO
		sTmp2:=	FCT_UPLOW_CASE(	xLowConvert:=TRUE,
								sInString:=ptrProfileList^[i].sName);
		IF sTmp = sTmp2 AND sTmp2 <> '' THEN RETURN; END_IF
	END_FOR

(* Confirm function *)
	xFctCtrleProfileName:=TRUE;
END_FUNCTION

(* POU GENERAL/FCT_UPLOW_CASE, ST *)
FUNCTION FCT_UPLOW_CASE : STRING
VAR_INPUT
	xLowConvert:BOOL;			(* FALSE=conversion to up case, TRUE=conversion in low case *)
	sInString:STRING;				(* string with 80 character, which will be convert *)
END_VAR
VAR
(* variable *)
	sListUpCase:STRING:='ABCDEFGHIJKLMNOPQRSTUVWXYZ';
	sListLowCase:STRING:='abcdefghijklmnopqrstuvwxyz';
	i:INT;
(* Tmp *)
	sTmp:STRING;
	iTmp:INT;
END_VAR
(****************************************************************************************************************************************************)
(***********                                                      This function convert a String in up or low case                                                                ************)
(****************************************************************************************************************************************************)
(* Init. *)
	FCT_UPLOW_CASE:='';

(*Test string size*)
	IF LEN(sInString) < 1 OR LEN(sInString) > 255 THEN RETURN; END_IF

	IF xLowConvert THEN
	(* Conversion to low case *)
		FOR i:= 1 TO LEN(sInString) DO
			sTmp:=MID(sInString,1,i);
			iTmp:=FIND(sListUpCase,sTmp);
			IF iTmp > 0 THEN FCT_UPLOW_CASE:=CONCAT(FCT_UPLOW_CASE,MID(sListLowCase,1,iTmp));
				ELSE FCT_UPLOW_CASE:=CONCAT(FCT_UPLOW_CASE,sTmp); END_IF
		END_FOR
	(* Conversion to up case *)
	ELSE
		FOR i:= 1 TO LEN(sInString) DO
			sTmp:=MID(sInString,1,i);
			iTmp:=FIND(sListLowCase,sTmp);
			IF iTmp > 0 THEN FCT_UPLOW_CASE:=CONCAT(FCT_UPLOW_CASE,MID(sListUpCase,1,iTmp));
				ELSE FCT_UPLOW_CASE:=CONCAT(FCT_UPLOW_CASE,sTmp); END_IF
		END_FOR
	END_IF
END_FUNCTION

(* POU PRG_VISU_LAYER5/FB_VISU/iFctExistProfileName, ST *)
FUNCTION iFctExistProfileName : INT
VAR_INPUT
	sProfileName:STRING(30);											(* name of the profile, which will be saved *)
	ptrProfileList:POINTER TO ARRAY[1..csiMaxProfile] OF ST_PROFILE_ID;	(* list of profil names which are saved *)
END_VAR
VAR
	i:INT;
	sTmp:STRING;
	sTmp2:STRING;
END_VAR
(****************************************************************************************************************************************************)
(***********                                               This Function check if the name of the profile already exists                                              ************)
(****************************************************************************************************************************************************)
(* Init. function *)
	iFctExistProfileName:=0;
	sTmp:=FCT_UPLOW_CASE(	xLowConvert:=TRUE,
							sInString:=sProfileName);

(* Search if name already exists *)
	FOR i:=1 TO csiMaxProfile DO
		sTmp2:=	FCT_UPLOW_CASE(	xLowConvert:=TRUE,
								sInString:=ptrProfileList^[i].sName);
		IF sTmp = sTmp2 AND sTmp2 <> '' THEN iFctExistProfileName:=i; RETURN; END_IF
	END_FOR
END_FUNCTION

(* POU PRG_VISU_LAYER5/FB_VISU/rFctCalcMaxToolDiameter, ST *)
FUNCTION rFctCalcMaxToolDiameter : REAL
VAR_INPUT
	rDistanceD1:REAL;		(* distance d1 of the prisma *)
	rDistanceD2:REAL;		(* distance d2 of the prisma *)
	rAnglePrism:REAL;		(* angle of the prisma *)
END_VAR
VAR
	rTmp: REAL;
	rTmpMaxDia: REAL;
END_VAR
(****************************************************************************************************************************************************)
(***********                    This Function calculate the maximum of the tooldiameter in case of the settled prisma                      ************)
(****************************************************************************************************************************************************)
rTmp:=SIN((90 - rAnglePrism/2) * PI/180);
IF rTmp <> 0 THEN
	rTmpMaxDia:=rDistanceD1/rTmp;
ELSE
	rTmpMaxDia:=0;
END_IF;
rFctCalcMaxToolDiameter:=rTmpMaxDia;
END_FUNCTION

(* POU PRG_VISU_LAYER5/FB_VISU/rFctCalcMinToolDiameter, ST *)
FUNCTION rFctCalcMinToolDiameter : REAL
VAR_INPUT
	rDistanceD1:REAL;		(* distance d1 of the prisma *)
	rDistanceD2:REAL;		(* distance d2 of the prisma *)
	rAnglePrism:REAL;		(* angle of the prisma *)
	bStateInputPrisma:BYTE;	(* choice of selected prisma *)
END_VAR
VAR
	rTmp: REAL;
	rTmp1: REAL;
	rMinD1_1: REAL;
	rMinD1_2: REAL;
	rReturnValue: REAL;
END_VAR
(****************************************************************************************************************************************************)
(***********                    This Function calculate the minimum of the tooldiameter in case of the settled prisma                      ************)
(****************************************************************************************************************************************************)
rFctCalcMinToolDiameter:=0;
rTmp:=TAN((rAnglePrism/2)*PI/180);
rTmp1:=SIN((rAnglePrism/2)*PI/180);
IF (rTmp <> 0) AND (rTmp1 <> 0) THEN
	rMinD1_1:=rDistanceD1/(rTmp * (1 + 1/rTmp1));
END_IF;
rMinD1_2:=rDistanceD2;
IF (bStateInputPrisma = 0) OR (bStateInputPrisma = 1) THEN
	IF (rMinD1_1 >= rMinD1_2) THEN
		rReturnValue:=rMinD1_1;
	ELSE
		rReturnValue:=rMinD1_2;
	END_IF;
ELSE
	rReturnValue:=rMinD1_1;
END_IF;
rFctCalcMinToolDiameter:=rReturnValue;
END_FUNCTION

(* POU PRG_VISU_LAYER5/FB_VISU/rFctCalcPrismaFactor, ST *)
FUNCTION rFctCalcPrismaFactor : REAL
VAR_INPUT
	rAnglePrism:REAL;	(* angle of the prisma *)
END_VAR
VAR
	rFactorPrisma: REAL;
END_VAR
(****************************************************************************************************************************************************)
(***********     This Function calculate the correctur factor for the GrindFeeder Axis dependent of the settled prisma         ************)
(****************************************************************************************************************************************************)
rFctCalcPrismaFactor:=0.0;
rFactorPrisma:=(1 + SIN((rAnglePrism / 2.0) * PI/180)) / (2.0 * SIN((rAnglePrism / 2.0) * PI / 180.0));
(* Auf 5 Kommastellen runden *)
rFactorPrisma:=	STRING_TO_REAL(	LREAL_TO_FMTSTR(	in:=rFactorPrisma,
														iPrecision:=5,
														bRound:=TRUE));

rFctCalcPrismaFactor:=rFactorPrisma;
END_FUNCTION

(* POU PRG_VISU_LAYER5/FB_VISU/FB_CTRLEBUTTON, ST *)
FUNCTION_BLOCK FB_CTRLEBUTTON
VAR_INPUT
	xHWStart:BOOL;							(* external start button *)
	xHWStop:BOOL;							(* external stop button *)
	dwActualPage:DWORD;					(* active number page of the visualisation *)
	T_VisuQVis:ST_QVIS;						(* data structure of the visualisation *)
	T_ExchgParam:ST_QVIS_EXCHG_PARAM;	(* data structure of the visualisation *)
	IxSafetyCircuitOn1:BOOL;					(* state of current if it is on or off from the channel 1 *)
	IxSafetyCircuitOn2:BOOL;					(* state of current if it is on or off from the channel 2 *)
END_VAR
VAR_OUTPUT
END_VAR
VAR_IN_OUT
	T_StartButton: ST_BUTTON;				(* data structure of the control button start *)
	T_StopButton:ST_BUTTON;				(* data structure of the control button stop *)
END_VAR
VAR
(* Init. variable *)
	xFirstExecution:BOOL:=FALSE;
(* Variable *)
	iIndexActivPage:INT;
	dwOldActualPage:DWORD;
(* FB Mask *)
	xMaskPageBtStart:BOOL;
	xMaskPageBtStop:BOOL;
(* Trigger *)
	RisingEdgeSignalStartButton:R_TRIG;
	RisingEdgeStartState:R_TRIG;
	RisingEdgeCfgBtStart:R_TRIG;
	RisingEdgeSignalStopButton:R_TRIG;
	RisingEdgeFlagStopProcess:R_TRIG;
(* Tmp variable *)
	xTmp:BOOL;
	(*RisingEdgeConfirmMessage: R_TRIG; *)
END_VAR
(****************************************************************************************************************************************************)
(***********             This Functionblock manage the external start and stop butto, also for the lamp of this button                  ************)
(****************************************************************************************************************************************************)
(* First execution *)
	IF NOT xFirstExecution THEN
		dwOldActualPage:=16#FFFFFFFF;
		RisingEdgeSignalStartButton(CLK:=FALSE);
		RisingEdgeStartState(CLK:=FALSE);
		RisingEdgeCfgBtStart(CLK:=FALSE);
		RisingEdgeSignalStopButton(CLK:=FALSE);
		RisingEdgeFlagStopProcess(CLK:=FALSE);
		(* Set first execution *)
		xFirstExecution:=TRUE;
	END_IF

(* exit FB if Qvis inactiv *)
	IF NOT(T_VisuQVis.T_CtrleVisu.xQvis) THEN RETURN; END_IF
	IF (dwActualPage < 1) OR (dwActualPage > 999) THEN RETURN; END_IF;

(* Index Activ Page *)
	IF dwActualPage = 0 THEN iIndexActivPage:=1;
	ELSE iIndexActivPage:=T_VisuQVis.T_PageIndex[dwActualPage].iIndexConfigPage; END_IF

(* Start Button *)
	xMaskPageBtStart:=FALSE;
	CASE dwActualPage OF
	(* Auto Geometry page *)
	10:	xTmp:=TRUE;
		IF xTmp AND (NOT(IxSafetyCircuitOn1) OR NOT(IxSafetyCircuitOn2)) THEN
			xTmp:=FALSE;	(* Energieversorgung muss eingeschaltet sein *)
		END_IF;
		IF xTmp AND ((T_ExchgParam.T_SafetyCtrl.bStateMessageError <> 0) OR (T_ExchgParam.T_SafetyCtrl.bStateMessageInfo <> 0)) THEN
			xTmp:=FALSE;
		END_IF;
		IF (T_ExchgParam.T_Visu.T_Message.iState = 401) OR (T_ExchgParam.T_Visu.T_Message.iState = 118) OR (T_ExchgParam.T_Visu.T_Message.iState = 119) OR (T_ExchgParam.T_Visu.T_Message.iState = 108) THEN
			xTmp:=FALSE;
		END_IF;
		(* copy state *)
		xMaskPageBtStart:=xTmp;
	(* Auto Groove page *)
	20:	xTmp:=TRUE;
		IF xTmp AND (NOT(IxSafetyCircuitOn1) OR NOT(IxSafetyCircuitOn2)) THEN
			xTmp:=FALSE;	(* Energieversorgung muss eingeschaltet sein *)
		END_IF;
		IF xTmp AND ((T_ExchgParam.T_SafetyCtrl.bStateMessageError <> 0) OR (T_ExchgParam.T_SafetyCtrl.bStateMessageInfo <> 0)) THEN
			xTmp:=FALSE;
		END_IF;
		IF (T_ExchgParam.T_Visu.T_Message.iState = 401) OR (T_ExchgParam.T_Visu.T_Message.iState = 118) OR (T_ExchgParam.T_Visu.T_Message.iState = 119) OR (T_ExchgParam.T_Visu.T_Message.iState = 108) THEN
			xTmp:=FALSE;
		END_IF;
		(* copy state *)
		xMaskPageBtStart:=xTmp;
	(* Reference page *)
	30:	xTmp:=TRUE;
		IF xTmp AND (NOT(IxSafetyCircuitOn1) OR NOT(IxSafetyCircuitOn2)) THEN
			xTmp:=FALSE;	(* Energieversorgung muss eingeschaltet sein *)
		END_IF;
		IF xTmp AND ((T_ExchgParam.T_SafetyCtrl.bStateMessageError <> 0) OR (T_ExchgParam.T_SafetyCtrl.bStateMessageInfo <> 0)) THEN
			xTmp:=FALSE;
		END_IF;
		IF (T_ExchgParam.T_Visu.T_Message.iState = 401) OR (T_ExchgParam.T_Visu.T_Message.iState = 118) OR (T_ExchgParam.T_Visu.T_Message.iState = 119) THEN
			xTmp:=FALSE;
		END_IF;
		IF (T_ExchgParam.T_StationCommon.iConfigMachineType = 1) THEN
			xTmp:=FALSE;
		END_IF;
		(* copy state *)
		xMaskPageBtStart:=xTmp;
	(* Tool Calibration page *)
	110:	xTmp:=TRUE;
		IF xTmp AND (NOT(IxSafetyCircuitOn1) OR NOT(IxSafetyCircuitOn2)) THEN
			xTmp:=FALSE;	(* Energieversorgung muss eingeschaltet sein *)
		END_IF;
		IF xTmp AND ((T_ExchgParam.T_SafetyCtrl.bStateMessageError <> 0) OR (T_ExchgParam.T_SafetyCtrl.bStateMessageInfo <> 0)) THEN
			xTmp:=FALSE;
		END_IF;
		IF (T_ExchgParam.T_Visu.T_Message.iState = 401) OR (T_ExchgParam.T_Visu.T_Message.iState = 118) OR (T_ExchgParam.T_Visu.T_Message.iState = 119) OR
		     (T_ExchgParam.T_Visu.T_Message.iState = 108) THEN
			xTmp:=FALSE;
		END_IF;
		IF ((T_ExchgParam.T_Machine.T_Process.wState AND 16#6) = 16#2) THEN
			xTmp:=FALSE;
		END_IF;
		IF T_ExchgParam.T_FunctionCommon.xOpenOverlayMeasureInput OR T_ExchgParam.T_FunctionCommon.xOpenOverlaySetGrindPlunge THEN
			xTmp:=FALSE;
		END_IF;
		(* copy state *)
		xMaskPageBtStart:=xTmp;
	(* Teach-in Tool Rotation page *)
	210:	xTmp:=	((T_ExchgParam.T_StationCommon.bStateMachine AND 16#7) = 16#1);
		IF xTmp AND (NOT(IxSafetyCircuitOn1) OR NOT(IxSafetyCircuitOn2)) THEN
			xTmp:=FALSE;	(* Energieversorgung muss eingeschaltet sein *)
		END_IF;
		IF xTmp AND ((T_ExchgParam.T_SafetyCtrl.bStateMessageError <> 0) OR (T_ExchgParam.T_SafetyCtrl.bStateMessageInfo <> 0)) THEN
			xTmp:=FALSE;
		END_IF;
		IF (T_ExchgParam.T_Visu.T_Message.iState = 401) OR (T_ExchgParam.T_Visu.T_Message.iState = 118) OR (T_ExchgParam.T_Visu.T_Message.iState = 119) OR
		     (T_ExchgParam.T_Visu.T_Message.iState = 101) THEN
			xTmp:=FALSE;
		END_IF;
		IF (T_ExchgParam.T_TeachIn.iSelectAxisToolRotation = 1) AND xTmp THEN
			IF ((T_ExchgParam.T_StationCommon.bStateAxisReelLeft AND 16#2) = 16#2) THEN
				xTmp:=FALSE;
			END_IF;
		END_IF;
		IF (T_ExchgParam.T_TeachIn.iSelectAxisToolRotation = 2) AND xTmp THEN
			IF ((T_ExchgParam.T_StationCommon.bStateAxisReelCenter AND 16#2) = 16#2) THEN
				xTmp:=FALSE;
			END_IF;
		END_IF;
		IF (T_ExchgParam.T_TeachIn.iSelectAxisToolRotation = 3) AND xTmp THEN
			IF ((T_ExchgParam.T_StationCommon.bStateAxisReelRight AND 16#2) = 16#2) THEN
				xTmp:=FALSE;
			END_IF;
		END_IF;
		(* copy state *)
		xMaskPageBtStart:=xTmp;
	(* Tool Torque page *)
	220:	xTmp:=	((T_ExchgParam.T_StationCommon.bStateMachine AND 16#7) = 16#1);
		IF xTmp AND (NOT(IxSafetyCircuitOn1) OR NOT(IxSafetyCircuitOn2)) THEN
			xTmp:=FALSE;	(* Energieversorgung muss eingeschaltet sein *)
		END_IF;
		IF xTmp AND ((T_ExchgParam.T_SafetyCtrl.bStateMessageError <> 0) OR (T_ExchgParam.T_SafetyCtrl.bStateMessageInfo <> 0)) THEN
			xTmp:=FALSE;
		END_IF;
		IF (T_ExchgParam.T_Visu.T_Message.iState = 401) OR (T_ExchgParam.T_Visu.T_Message.iState = 118) OR (T_ExchgParam.T_Visu.T_Message.iState = 119) OR
		     (T_ExchgParam.T_Visu.T_Message.iState = 101) THEN
			xTmp:=FALSE;
		END_IF;
		IF ((T_ExchgParam.T_StationCommon.bStateAxisReelLeft AND 16#2) = 16#2) THEN
			xTmp:=FALSE;
		END_IF;
		(* copy state *)
		xMaskPageBtStart:=xTmp;
	(* Teach-in Tool Feeder page *)
	310:	xTmp:=	xTmp:=	((T_ExchgParam.T_StationCommon.bStateMachine AND 16#7) = 16#1);
		IF xTmp AND (NOT(IxSafetyCircuitOn1) OR NOT(IxSafetyCircuitOn2)) THEN
			xTmp:=FALSE;	(* Energieversorgung muss eingeschaltet sein *)
		END_IF;
		IF xTmp AND ((T_ExchgParam.T_SafetyCtrl.bStateMessageError <> 0) OR (T_ExchgParam.T_SafetyCtrl.bStateMessageInfo <> 0)) THEN
			xTmp:=FALSE;
		END_IF;
		IF (T_ExchgParam.T_Visu.T_Message.iState = 401) OR (T_ExchgParam.T_Visu.T_Message.iState = 118) OR (T_ExchgParam.T_Visu.T_Message.iState = 119) OR
		     (T_ExchgParam.T_Visu.T_Message.iState = 101) OR (T_ExchgParam.T_Visu.T_Message.iState = 18) THEN
			xTmp:=FALSE;
		END_IF;
		IF (T_ExchgParam.T_TeachIn.iSelectAxisWireFeeder = 1) AND xTmp THEN
			IF ((T_ExchgParam.T_StationCommon.bStateAxisWireFeeder AND 16#2) = 16#2) THEN
				xTmp:=FALSE;
			END_IF;
		END_IF;
		(* copy state *)
		xMaskPageBtStart:=xTmp;
	(* Teach-in Tool Feeder page *)
	330:	xTmp:=	xTmp:=	((T_ExchgParam.T_StationCommon.bStateMachine AND 16#7) = 16#1);
		IF xTmp AND (NOT(IxSafetyCircuitOn1) OR NOT(IxSafetyCircuitOn2)) THEN
			xTmp:=FALSE;	(* Energieversorgung muss eingeschaltet sein *)
		END_IF;
		IF xTmp AND ((T_ExchgParam.T_SafetyCtrl.bStateMessageError <> 0) OR (T_ExchgParam.T_SafetyCtrl.bStateMessageInfo <> 0)) THEN
			xTmp:=FALSE;
		END_IF;
		IF (T_ExchgParam.T_Visu.T_Message.iState = 401) OR (T_ExchgParam.T_Visu.T_Message.iState = 118) OR (T_ExchgParam.T_Visu.T_Message.iState = 119) OR
		     (T_ExchgParam.T_Visu.T_Message.iState = 101) OR (T_ExchgParam.T_Visu.T_Message.iState = 18) THEN
			xTmp:=FALSE;
		END_IF;
		IF (T_ExchgParam.T_TeachIn.iSelectAxisWireFeeder = 1) AND xTmp THEN
			IF ((T_ExchgParam.T_StationCommon.bStateAxisWireFeeder AND 16#2) = 16#2) THEN
				xTmp:=FALSE;
			END_IF;
		END_IF;
		(* copy state *)
		xMaskPageBtStart:=xTmp;
	(* Teach-in Grind Feeder page *)
	410:	xTmp:=	xTmp:=	((T_ExchgParam.T_StationCommon.bStateMachine AND 16#7) = 16#1);
		IF xTmp AND (NOT(IxSafetyCircuitOn1) OR NOT(IxSafetyCircuitOn2)) THEN
			xTmp:=FALSE;	(* Energieversorgung muss eingeschaltet sein *)
		END_IF;
		IF xTmp AND ((T_ExchgParam.T_SafetyCtrl.bStateMessageError <> 0) OR (T_ExchgParam.T_SafetyCtrl.bStateMessageInfo <> 0)) THEN
			xTmp:=FALSE;
		END_IF;
		IF (T_ExchgParam.T_Visu.T_Message.iState = 401) OR (T_ExchgParam.T_Visu.T_Message.iState = 118) OR (T_ExchgParam.T_Visu.T_Message.iState = 119) OR
		     (T_ExchgParam.T_Visu.T_Message.iState = 101) THEN
			xTmp:=FALSE;
		END_IF;
		IF (T_ExchgParam.T_TeachIn.iSelectAxisGrind = 1) AND xTmp THEN
			IF ((T_ExchgParam.T_StationCommon.bStateAxisGrind AND 16#2) = 16#2) THEN
				xTmp:=FALSE;
			END_IF;
		END_IF;
		(* copy state *)
		xMaskPageBtStart:=xTmp;
	END_CASE

	(* Set state button start *)
	RisingEdgeSignalStartButton(CLK:=xHWStart);
	IF RisingEdgeSignalStartButton.Q THEN T_StartButton.xInputState:=TRUE; ELSE T_StartButton.xInputState:=FALSE; END_IF
	T_StartButton.xInputState:=T_StartButton.xInputState AND T_VisuQVis.T_ConfigPage[iIndexActivPage].xMaskBtStart;

	(* if page change => init. trigger *)
	IF dwActualPage <> dwOldActualPage THEN
		RisingEdgeStartState(CLK:=FALSE);
		RisingEdgeCfgBtStart(CLK:=FALSE);
		(* save value *)
		dwOldActualPage:=dwActualPage;
	END_IF

	(* Led off if action is starting *)
	RisingEdgeStartState(CLK:=T_StartButton.xInputState);
	IF RisingEdgeStartState.Q THEN T_StartButton.xLedState:=FALSE; END_IF
	RisingEdgeCfgBtStart(CLK:=xMaskPageBtStart);
	IF RisingEdgeCfgBtStart.Q THEN T_StartButton.xLedState:=TRUE; END_IF
	T_StartButton.xLedState:=T_StartButton.xLedState AND T_VisuQVis.T_ConfigPage[iIndexActivPage].xMaskBtStart;

	(* set page mask *)
	T_StartButton.xInputState:=T_StartButton.xInputState AND xMaskPageBtStart;
	T_StartButton.xLedState:=T_StartButton.xLedState AND xMaskPageBtStart;

(* Stop Button *)
	xMaskPageBtStop:=FALSE;
	RisingEdgeSignalStopButton(CLK:=xHWStop);
	IF RisingEdgeSignalStopButton.Q THEN T_StopButton.xInputState:=TRUE; ELSE T_StopButton.xInputState:=FALSE; END_IF
	T_StopButton.xInputState:=T_StopButton.xInputState AND T_VisuQVis.T_ConfigPage[iIndexActivPage].xMaskBtStop;
	T_StopButton.xLedState:=T_VisuQVis.T_ConfigPage[iIndexActivPage].xMaskBtStop;

	(* if machine process inactiv => set mask inactiv *)
	IF dwActualPage > 0 THEN
		IF (T_ExchgParam.T_Machine.T_Process.wState AND 16#14) = 16#0 THEN
		(* process activ and no error *)
			IF (T_ExchgParam.T_Machine.T_Process.wState AND 16#80) = 16#0 THEN xMaskPageBtStop:=TRUE; ELSE xMaskPageBtStop:=FALSE; END_IF
		ELSIF ((dwActualPage = 210) OR (dwActualPage = 310) OR (dwActualPage = 410)) THEN
			(* Achse muss Aktiv sein, Stationsendflag muss gesetzt sein, Prozessendflag muss gesetzt sein *)
			IF ((T_ExchgParam.T_StationCommon.bStateMachine AND 16#7) = 16#3) AND ((T_ExchgParam.T_Machine.T_Process.wState AND 16#2) = 16#0) THEN
				xMaskPageBtStop:=TRUE;
			END_IF;
			(* Achse darf nicht Aktiv sein, Stationsendflag muss gesetzt sein,  Prozessendflag muss gesetzt sein *)
			IF ((T_ExchgParam.T_StationCommon.bStateMachine AND 16#7) = 16#1) AND ((T_ExchgParam.T_Machine.T_Process.wState AND 16#2) = 16#0) THEN
				xMaskPageBtStop:=FALSE;
				IF (T_ExchgParam.T_TeachIn.iSelectAxisToolRotation = 1) AND (dwActualPage = 210) THEN
					IF ((T_ExchgParam.T_StationCommon.bStateAxisReelLeft AND 16#2) = 16#2) THEN
						xMaskPageBtStop:=TRUE;
					END_IF;
				END_IF;
				IF (T_ExchgParam.T_TeachIn.iSelectAxisToolRotation = 2) AND (dwActualPage = 210) THEN
					IF ((T_ExchgParam.T_StationCommon.bStateAxisReelCenter AND 16#2) = 16#2) THEN
						xMaskPageBtStop:=TRUE;
					END_IF;
				END_IF;
				IF (T_ExchgParam.T_TeachIn.iSelectAxisToolRotation = 3) AND (dwActualPage = 210) THEN
					IF ((T_ExchgParam.T_StationCommon.bStateAxisReelRight AND 16#2) = 16#2) THEN
						xMaskPageBtStop:=TRUE;
					END_IF;
				END_IF;
				IF (T_ExchgParam.T_TeachIn.iSelectAxisWireFeeder = 1) AND (dwActualPage = 310) THEN
					IF ((T_ExchgParam.T_StationCommon.bStateAxisWireFeeder AND 16#2) = 16#2) THEN
						xMaskPageBtStop:=TRUE;
					END_IF;
				END_IF;
				IF (T_ExchgParam.T_TeachIn.iSelectAxisGrind = 1) AND (dwActualPage = 410) THEN
					IF ((T_ExchgParam.T_StationCommon.bStateAxisGrind AND 16#2) = 16#2) THEN
						xMaskPageBtStop:=TRUE;
					END_IF;
				END_IF;
			END_IF;
			IF (T_VisuQVis.T_CtrleAction.iFunction = 301) AND NOT(T_VisuQVis.T_CtrleAction.xDone) THEN
				xMaskPageBtStop:=FALSE;
			END_IF;
		ELSIF (dwActualPage = 220) THEN
			(* Achse muss Aktiv sein, Stationsendflag muss gesetzt sein, Prozessendflag muss gesetzt sein *)
			xMaskPageBtStop:=FALSE;
			IF ((T_ExchgParam.T_StationCommon.bStateAxisReelLeft AND 16#2) = 16#2) THEN
				xMaskPageBtStop:=TRUE;
			END_IF;
			IF (T_VisuQVis.T_CtrleAction.iFunction = 403) AND NOT(T_VisuQVis.T_CtrleAction.xDone) THEN
				xMaskPageBtStop:=FALSE;
			END_IF;
		(* process inactiv *)
		ELSE xMaskPageBtStop:=FALSE; END_IF
		IF (T_ExchgParam.T_Visu.T_Message.iState = 401) OR (T_ExchgParam.T_Visu.T_Message.iState = 118) OR (T_ExchgParam.T_Visu.T_Message.iState = 119) THEN
			xMaskPageBtStop:=FALSE;
		END_IF;
		IF NOT(IxSafetyCircuitOn1) OR NOT(IxSafetyCircuitOn2) THEN
			xMaskPageBtStop:=FALSE;
		END_IF;
	END_IF

	(* set page mask *)
	T_StopButton.xInputState:=T_StopButton.xInputState AND xMaskPageBtStop;
	T_StopButton.xLedState:=T_StopButton.xLedState AND xMaskPageBtStop;
END_FUNCTION_BLOCK

(* POU PRG_PROCESS_LAYER4/PRG_PROCESS, FBD *)
PROGRAM PRG_PROCESS
VAR
	FBProcess: FB_PROCESS;
	xReady: BOOL;
	xEnd: BOOL;
	xStop: BOOL;
	xReferenced: BOOL;
	xError: BOOL;
	iErrorNr: DINT;
	iFunctionNr: INT;
END_VAR
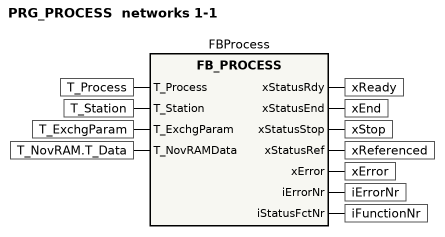
_FBD_ (* Function Block Diagram *)
NETWORK 1 (* PROCESS LEVEL-->LAYER 4 *)
	FBProcess:FB_PROCESS(T_Process: T_Process, T_Station: T_Station, T_ExchgParam: T_ExchgParam, T_NovRAMData: T_NovRAM.T_Data, xStatusEnd => xEnd, xStatusStop => xStop, xStatusRef => xReferenced, xError => xError, iErrorNr => iErrorNr, iStatusFctNr => iFunctionNr) => xReady
_END_FBD_
(* the same logic as Structured Text *)
(* Network 1: PROCESS LEVEL-->LAYER 4 *)
FBProcess(T_Process := T_Process, T_Station := T_Station, T_ExchgParam := T_ExchgParam, T_NovRAMData := T_NovRAM.T_Data);
xEnd := FBProcess.xStatusEnd;
xStop := FBProcess.xStatusStop;
xReferenced := FBProcess.xStatusRef;
xError := FBProcess.xError;
iErrorNr := FBProcess.iErrorNr;
iFunctionNr := FBProcess.iStatusFctNr;
xReady := FBProcess.xStatusRdy;
END_PROGRAM

(* POU GENERAL/FB_PROCESS, ST *)
FUNCTION_BLOCK FB_PROCESS
VAR_INPUT
END_VAR
VAR_IN_OUT
	T_Process : ST_PROCESS;				(* data structure of the processlevel *)
	T_Station : ST_STATION;					(* data structure of the stationlevel *)
	T_ExchgParam:ST_QVIS_EXCHG_PARAM;	(* data structure of the visualisation *)
	T_NovRAMData:ST_DATA_RETAIN;		(* data structure of the NovRam *)
END_VAR
VAR_OUTPUT
	xStatusRdy : BOOL := FALSE;				(* state of the processlevel if it is ready or not *)
	xStatusEnd : BOOL := FALSE;				(* state of the processlevel if a process is active or not *)
	xStatusStop : BOOL := FALSE;				(* state of the processlevel if a process will be stopped *)
	xStatusRef : BOOL := FALSE;				(* state of the processlevel if the machine is referenced *)
	xError : BOOL := FALSE;					(* state of the processlevel if the machine has an error *)
	iErrorNr : DINT :=0;							(* state of the processlevel if the machine has an error, in this case it will give the errornumber *)
	iStatusFctNr : INT := 0;						(* state of the processlevel, which process is active *)
END_VAR
VAR
	xStartFunction: BOOL;
	xSetEnd: BOOL;
	iPrcFunctionNr: INT;
	xProcessError: BOOL;
	xInitError: BOOL;
	xTmpStart: BOOL;
	xInitStart: BOOL;
	xInitStop: BOOL;
	xTmpStopFunction: BOOL;
	xDisable: BOOL;
	xResetRef: BOOL;
	xInitStopCycle: BOOL;
	xTmpStopCycleFunction: BOOL;
(* end modif test torque *)
	FBErrorMessage : FB_ErrorMessage;
	FBPrcMachineReference: FB_PrcMachineReference;
	FBPrcAutoGeometry: FB_PrcAutoGeometry;
	diTmpErrorNr: DINT;
	xResetAutoGeometry: BOOL;
	FBPrcAutoGroove: FB_PrcAutoGroove;
	xResetAutoGroove: BOOL;
	FBPrcToolCalibration: FB_PrcToolCalibration;
	xResetToolCalibration: BOOL;
END_VAR
(****************************************************************************************************************************************************)
(***********                                            This Functionblock manage all the machine process                                                             ************)
(****************************************************************************************************************************************************)
IF NOT(T_Process.xEnable) THEN
	T_Process.xRdy:=FALSE;
	xDisable:=TRUE;
	RETURN;
ELSE
	IF xDisable THEN
		T_Process.xRdy:=TRUE;
		xDisable:=FALSE;
		xSetEnd:=TRUE;
	END_IF;
END_IF;
(******************************************************************************************************************************************)
(****************************				                  Status Part                                                            *****************************)
(******************************************************************************************************************************************)
xStatusRdy:=T_Process.xRdy;
xStatusEnd:=T_Process.xEnd;
xStatusRef:=T_Station.TControl.xReferenced;
T_Process.xReferenced:=xStatusRef;
xError:=T_Process.xError;
iStatusFctNr:=iPrcFunctionNr;


(******************************************************************************************************************************************)
(****************************				         Error Controlling Part                                                  *****************************)
(******************************************************************************************************************************************)
IF xProcessError OR (T_Process.TFctProcess.xError AND T_Process.xRdy AND NOT(xSetEnd)) THEN
	IF NOT(xInitError) THEN
		xInitError:=TRUE;
		xProcessError:=TRUE;
		T_Process.TFctProcess.xQuitErr:=TRUE;
		T_Process.xProcessHold:=FALSE;
		diTmpErrorNr:=T_Process.TFctProcess.diErrorNr;
	END_IF;
	IF NOT(T_Process.TFctProcess.xQuitErr) AND T_Process.TFctProcess.xEnd AND (T_Process.diErrorNr = 0)THEN
		FBErrorMessage(	diErrorNr:=diTmpErrorNr,
						T_ErrorList:=T_ErrorList);
		T_ExchgParam.T_Visu.T_Message.sDynamicTextEnglish:=FBErrorMessage.sErrorTextEnglish;
		T_ExchgParam.T_Visu.T_Message.sDynamicTextDeutsch:=FBErrorMessage.sErrorTextDeutsch;
		T_ExchgParam.T_Visu.T_Message.sDynamicTextFrancais:=FBErrorMessage.sErrorTextFrancais;
		T_Process.diErrorNr:=diTmpErrorNr;
		T_Process.xError:=TRUE;
	END_IF;
	IF T_Process.xQuitError AND NOT(T_Process.TFctProcess.xQuitErr) THEN
		T_Process.xProcessHold:=FALSE;
		T_ExchgParam.T_Visu.T_Message.sDynamicTextEnglish:='';
		T_ExchgParam.T_Visu.T_Message.sDynamicTextDeutsch:='';
		T_ExchgParam.T_Visu.T_Message.sDynamicTextFrancais:='';
		xInitError:=FALSE;
		T_Process.xQuitError:=FALSE;
		xSetEnd:=TRUE;
	END_IF;
END_IF;
(******************************************************************************************************************************************)
(****************************				         Main Controlling Part                                                  *****************************)
(******************************************************************************************************************************************)
IF (T_Process.xStart OR xTmpStart) AND T_Process.xRdy AND NOT(xSetEnd) THEN
	IF NOT(xInitStart) THEN
		xInitStart:=TRUE;
		xTmpStart:=TRUE;
		T_Process.xStop:=FALSE;
		T_Process.xStopCycle:=FALSE;
		T_Process.xStart:=FALSE;
		T_Process.xEnd:=FALSE;
		T_Process.xProcessHold:=FALSE;
		T_Process.TFctProcess.xStart:=TRUE;
		xStartFunction:=TRUE;
		iPrcFunctionNr:=T_Process.iFunctNr;
	END_IF;
	IF T_Process.xAbord AND (T_Process.xStopCycle OR T_Process.xStop) THEN
		T_Process.xStopCycle:=T_Process.xStop:=FALSE;		(* Prozess ist am abbrechen, diese Flag können nicht mehr berücksichtigt werden *)
	END_IF;
	IF T_Process.xStopCycle THEN
		IF NOT(xInitStopCycle) THEN
			xInitStopCycle:=TRUE;
			T_Process.TFctProcess.xStopCycle:=TRUE;
		END_IF;
		IF NOT(T_Process.TFctProcess.xStopCycle) AND T_Process.TFctProcess.xProcessHold THEN
			xInitStopCycle:=FALSE;
			T_Process.xStopCycle:=FALSE;
			T_Process.xProcessHold:=TRUE;
			xTmpStopCycleFunction:=TRUE;
		END_IF;
		IF NOT(T_Process.TFctProcess.xStopCycle) AND NOT(T_Process.TFctProcess.xProcessHold) THEN
			xInitStopCycle:=FALSE;
			T_Process.xStopCycle:=FALSE;
			T_Process.xProcessHold:=FALSE;
			xTmpStopCycleFunction:=FALSE;
		END_IF;
	END_IF;
	IF T_Process.xStop THEN
		IF NOT(xInitStop) THEN
			xInitStop:=TRUE;
			T_Process.TFctProcess.xStop:=TRUE;
		END_IF;
		IF NOT(T_Process.TFctProcess.xStop) AND T_Process.TFctProcess.xProcessHold THEN
			xInitStop:=FALSE;
			T_Process.xProcessHold:=TRUE;
			T_Process.xStop:=FALSE;
			xTmpStopFunction:=TRUE;
		END_IF;
		IF NOT(T_Process.TFctProcess.xStop) AND NOT(T_Process.TFctProcess.xProcessHold) THEN
			xInitStop:=FALSE;
			T_Process.xStop:=FALSE;
			T_Process.xProcessHold:=FALSE;
			xTmpStopFunction:=FALSE;
		END_IF;
	END_IF;
	IF T_Process.xStart AND (xTmpStopFunction OR xTmpStopCycleFunction) AND NOT(T_Process.xAbord) THEN
		T_Process.xStart:=T_Process.xProcessHold:=FALSE;
		xTmpStopFunction:=FALSE;
		xTmpStopCycleFunction:=FALSE;
		T_Process.TFctProcess.xStart:=TRUE;
	END_IF;
	IF T_Process.xAbord AND (xTmpStopFunction OR xTmpStopCycleFunction) THEN
		T_Process.xProcessHold:=FALSE;
		T_Process.xStart:=FALSE;
		xTmpStopFunction:=FALSE;
		xTmpStopCycleFunction:=FALSE;
		T_Process.TFctProcess.xAbord:=TRUE;
	END_IF;
	IF NOT(T_Process.TFctProcess.xStart) AND T_Process.TFctProcess.xEnd AND NOT(xProcessError) THEN
		xTmpStart:=FALSE;
		xInitStart:=FALSE;
		xSetEnd:=TRUE;
	END_IF;
END_IF;
(******************************************************************************************************************************************)
(****************************				              Funktionen                                                               *****************************)
(******************************************************************************************************************************************)
IF xStartFunction AND NOT(xSetEnd) THEN
	IF (iPrcFunctionNr = 10) THEN
	(* Process AutoGeometry *)
		FBPrcAutoGeometry(	xMicroRodActive:=(T_NovRAMData.T_Standard.T_MachineConfig.iConfigMachineType = 2),
							xBeckhoffDriveActive:=(T_NovRAMData.T_Standard.T_MachineConfig.iConfigAxisType = 2),
							xStart:=T_Process.TFctProcess.xStart ,
							xStop:=T_Process.TFctProcess.xStop ,
							xStopCycle:=T_Process.TFctProcess.xStopCycle,
							xQuitErr:=T_Process.TFctProcess.xQuitErr ,
							xAbord:=T_Process.TFctProcess.xAbord ,
							T_Station:= T_Station,
							T_Process:= T_Process,
							xReset:= xResetAutoGeometry,
							T_ExchgParam:= T_ExchgParam,
							T_NovRAMData:=T_NovRAMData,
							xEnd=>T_Process.TFctProcess.xEnd ,
							xError=>T_Process.TFctProcess.xError ,
							diErrorNr=>T_Process.TFctProcess.diErrorNr);
	END_IF;
	IF (iPrcFunctionNr = 20) THEN
	(* Process AutoGroove *)
		FBPrcAutoGroove(	xMicroRodActive:=(T_NovRAMData.T_Standard.T_MachineConfig.iConfigMachineType = 2),
							xBeckhoffDriveActive:=(T_NovRAMData.T_Standard.T_MachineConfig.iConfigAxisType = 2),
							xStart:=T_Process.TFctProcess.xStart ,
							xStop:=T_Process.TFctProcess.xStop ,
							xQuitErr:=T_Process.TFctProcess.xQuitErr ,
							xAbord:=T_Process.TFctProcess.xAbord ,
							T_Station:= T_Station,
							T_Process:= T_Process,
							xReset:= xResetAutoGroove,
							T_ExchgParam:= T_ExchgParam,
							xDoNotMoveGrindPosition:=T_NovRAMData.T_ProcessImageData.T_AutoGroovePara.xBlockGrindFeeder,
							xPlungeActive:=T_NovRAMData.T_ProcessImageData.T_AutoGroovePara.xPlungeActivationGroove,
							T_NovRAMData:=T_NovRAMData,
							xEnd=>T_Process.TFctProcess.xEnd ,
							xError=>T_Process.TFctProcess.xError ,
							diErrorNr=>T_Process.TFctProcess.diErrorNr);
	END_IF;
	IF (iPrcFunctionNr = 30) THEN
	(* Process Machine Reference *)
		FBPrcMachineReference(	xMicroRodActive:=(T_NovRAMData.T_Standard.T_MachineConfig.iConfigMachineType = 2),
								xBeckhoffDriveActive:=(T_NovRAMData.T_Standard.T_MachineConfig.iConfigAxisType = 2),
								xStart:=T_Process.TFctProcess.xStart ,
								xStop:=T_Process.TFctProcess.xStop ,
								xQuitErr:=T_Process.TFctProcess.xQuitErr ,
								xAbord:=T_Process.TFctProcess.xAbord ,
								T_Station:= T_Station,
								T_Process:= T_Process,
								xReset:= xResetRef,
								T_ExchgParam:= T_ExchgParam,
								T_NovRAMData:=T_NovRAMData,
								xEnd=>T_Process.TFctProcess.xEnd ,
								xError=>T_Process.TFctProcess.xError ,
								diErrorNr=>T_Process.TFctProcess.diErrorNr);
	END_IF;
	IF (iPrcFunctionNr = 40) THEN
	(* Process ToolCalibration *)
		FBPrcToolCalibration(	xMicroRodActive:=(T_NovRAMData.T_Standard.T_MachineConfig.iConfigMachineType = 2),
							xBeckhoffDriveActive:=(T_NovRAMData.T_Standard.T_MachineConfig.iConfigAxisType = 2),
							xStart:=T_Process.TFctProcess.xStart ,
							xStop:=T_Process.TFctProcess.xStop ,
							xQuitErr:=T_Process.TFctProcess.xQuitErr ,
							xAbord:=T_Process.TFctProcess.xAbord ,
							T_Station:= T_Station,
							T_Process:= T_Process,
							xReset:= xResetAutoGeometry,
							T_ExchgParam:= T_ExchgParam,
							T_NovRAMData:=T_NovRAMData,
							xEnd=>T_Process.TFctProcess.xEnd ,
							xError=>T_Process.TFctProcess.xError ,
							diErrorNr=>T_Process.TFctProcess.diErrorNr);
	END_IF;
END_IF;
(******************************************************************************************************************************************)
(****************************				         Init / Reset Hardware                                                 *****************************)
(******************************************************************************************************************************************)
IF xSetEnd THEN
	xStartFunction:=FALSE;
	xProcessError:=FALSE;
	xInitError:=FALSE;
	xInitStart:=FALSE;
	xInitStop:=FALSE;
	xSetEnd:=FALSE;
	xTmpStart:=FALSE;
	T_Process.xEnd:=TRUE;
	T_Process.xStart:=FALSE;
	T_Process.xStop:=FALSE;
	T_Process.xError:=FALSE;
	T_Process.diErrorNr:=0;
	T_Process.xAbord:=FALSE;
	T_Process.xQuitError:=FALSE;
	T_Process.wStatus:=0;
	T_Process.xAbord:=FALSE;
	T_Process.xStopCycle:=FALSE;
	T_Process.xProcessHold:=FALSE;
	xResetRef:=TRUE;
	FBPrcMachineReference(	xStart:=T_Process.TFctProcess.xStart ,
							xStop:=T_Process.TFctProcess.xStop ,
							xQuitErr:=T_Process.TFctProcess.xQuitErr ,
							xAbord:=T_Process.TFctProcess.xAbord ,
							T_Station:= T_Station,
							T_Process:= T_Process,
							xReset:= xResetRef,
							T_ExchgParam:= T_ExchgParam,
							xEnd=>T_Process.TFctProcess.xEnd ,
							xError=>T_Process.TFctProcess.xError ,
							diErrorNr=>T_Process.TFctProcess.diErrorNr);
	xResetAutoGeometry:=TRUE;
	FBPrcAutoGeometry(	xMicroRodActive:=(T_NovRAMData.T_Standard.T_MachineConfig.iConfigMachineType = 2),
						xBeckhoffDriveActive:=(T_NovRAMData.T_Standard.T_MachineConfig.iConfigAxisType = 2),
						xStart:=T_Process.TFctProcess.xStart ,
						xStop:=T_Process.TFctProcess.xStop ,
						xStopCycle:=T_Process.TFctProcess.xStopCycle,
						xQuitErr:=T_Process.TFctProcess.xQuitErr ,
						xAbord:=T_Process.TFctProcess.xAbord ,
						T_Station:= T_Station,
						T_Process:= T_Process,
						xReset:= xResetAutoGeometry,
						T_ExchgParam:= T_ExchgParam,
						T_NovRAMData:=T_NovRAMData,
						xEnd=>T_Process.TFctProcess.xEnd ,
						xError=>T_Process.TFctProcess.xError ,
						diErrorNr=>T_Process.TFctProcess.diErrorNr);
	xResetAutoGroove:=TRUE;
	FBPrcAutoGroove(	xMicroRodActive:=(T_NovRAMData.T_Standard.T_MachineConfig.iConfigMachineType = 2),
						xBeckhoffDriveActive:=(T_NovRAMData.T_Standard.T_MachineConfig.iConfigAxisType = 2),
						xStart:=T_Process.TFctProcess.xStart ,
						xStop:=T_Process.TFctProcess.xStop ,
						xQuitErr:=T_Process.TFctProcess.xQuitErr ,
						xAbord:=T_Process.TFctProcess.xAbord ,
						T_Station:= T_Station,
						T_Process:= T_Process,
						xReset:= xResetAutoGroove,
						T_ExchgParam:= T_ExchgParam,
						xDoNotMoveGrindPosition:=T_NovRAMData.T_ProcessImageData.T_AutoGroovePara.xBlockGrindFeeder,
						xPlungeActive:=T_NovRAMData.T_ProcessImageData.T_AutoGroovePara.xPlungeActivationGroove,
						T_NovRAMData:=T_NovRAMData,
						xEnd=>T_Process.TFctProcess.xEnd ,
						xError=>T_Process.TFctProcess.xError ,
						diErrorNr=>T_Process.TFctProcess.diErrorNr);
	xResetToolCalibration:=TRUE;
	FBPrcToolCalibration(	xMicroRodActive:=(T_NovRAMData.T_Standard.T_MachineConfig.iConfigMachineType = 2),
						xBeckhoffDriveActive:=(T_NovRAMData.T_Standard.T_MachineConfig.iConfigAxisType = 2),
						xStart:=T_Process.TFctProcess.xStart ,
						xStop:=T_Process.TFctProcess.xStop ,
						xQuitErr:=T_Process.TFctProcess.xQuitErr ,
						xAbord:=T_Process.TFctProcess.xAbord ,
						T_Station:= T_Station,
						T_Process:= T_Process,
						xReset:= xResetToolCalibration,
						T_ExchgParam:= T_ExchgParam,
						T_NovRAMData:=T_NovRAMData,
						xEnd=>T_Process.TFctProcess.xEnd ,
						xError=>T_Process.TFctProcess.xError ,
						diErrorNr=>T_Process.TFctProcess.diErrorNr);
END_IF;
END_FUNCTION_BLOCK

(* POU PRG_PROCESS_LAYER4/FB_PROCESS/FB_PrcMachineReference, ST *)
FUNCTION_BLOCK FB_PrcMachineReference
VAR_INPUT
	xMicroRodActive: BOOL;				(* choice of the machine MicroWire or MicroRod *)
	xBeckhoffDriveActive: BOOL;			(* choice of the axis Beckhoff or EcoStep *)
	T_NovRAMData:ST_DATA_RETAIN;	(* Novram structure for all Machine parameter *)
END_VAR
VAR_IN_OUT
	xStart : BOOL;							(* start a process *)
	xStop : BOOL;							(* stop a process *)
	xQuitErr : BOOL;						(* quit an error *)
	xAbord : BOOL;						(* abord a process *)
	T_Station : ST_STATION;				(* data structure of the stationlevel *)
	T_Process : ST_PROCESS;			(* data strucuture of the processlevel *)
	xReset : BOOL;						(* reset the FB *)
	T_ExchgParam:ST_QVIS_EXCHG_PARAM;	(* data structure of the visualisation *)
END_VAR
VAR_OUTPUT
	xEnd : BOOL;							(* Endflag of the process *)
	xError : BOOL;							(* Errorflag of the process *)
	diErrorNr : DINT;						(* Error number of the process *)
END_VAR
VAR
	iStepPrc: INT;
	xInitStep: BOOL;
	xSetError: BOOL;
	xSetEnd: BOOL;
	xStartMainCtr: BOOL;
	xStartMainPrc: BOOL;
	xInitMainCtr: BOOL;
	xFreeze: BOOL;
	xInitError: BOOL;
	iStepError: INT;
	xTmpStop: BOOL;
	xSetTmpError: BOOL;
	xTmpAbord: BOOL;
	diTmpErrNr: DINT;
	xSetEndPrc : BOOL;
	iTmpFunctionNr:INT;
	xStopFctStation1: BOOL;
	iStepStop: INT;
	iTmpStationFunctionNr: INT;
	xStartProcess: BOOL;
	TONStartTimer: TON;
	tStepTime: TIME;
	TONStartTimer1: TON;
END_VAR
(****************************************************************************************************************************************************)
(***********   This Functionblock define the process for the Machine referencing-->it is needed only for the MicroRod     ************)
(****************************************************************************************************************************************************)

(******************************************************************************************************************************************)
(****************************				           Reset Function Part                                                 *****************************)
(******************************************************************************************************************************************)
IF xReset THEN
	xReset:=FALSE;
	xSetEnd:=TRUE;
END_IF;
(******************************************************************************************************************************************)
(****************************				              Error Controlling Part                                            *****************************)
(******************************************************************************************************************************************)
IF (xSetError OR T_Station.TControl.xError) AND NOT(xSetEnd) THEN
	IF NOT(xInitError) THEN
		iStepError:=100;
		xInitError:=TRUE;
		IF NOT(xSetError) THEN
			xSetError:=TRUE;
			xSetTmpError:=FALSE;
		ELSE
			xSetTmpError:=TRUE;
		END_IF;
	END_IF;
	CASE iStepError OF
		100:	IF T_Station.TControl.xError THEN
				diErrorNr:=T_Station.TControl.diErrorNr;
			END_IF;
			IF xSetTmpError THEN
				diErrorNr:=diTmpErrNr;
			END_IF;
			iStepError:=200;
		200:	IF xSetTmpError THEN
				xSetTmpError:=FALSE;
				xStopFctStation1:=FALSE;
				iStepError:=300;
			ELSE
				IF NOT(T_Station.TControl.xError) AND NOT(T_Station.TControl.xEnd) THEN
					IF (T_Station.TControl.iFunctNr = 1) THEN
						T_Station.TControl.xStop:=TRUE;
						xStopFctStation1:=TRUE;
					ELSE
						xStopFctStation1:=FALSE;
					END_IF;
				END_IF;
				iStepError:=300;
			END_IF;
		300:	IF xStopFctStation1 THEN
				IF NOT(T_Station.TControl.xStop) THEN
					xStopFctStation1:=FALSE;
				END_IF;
			END_IF;
			IF NOT(xStopFctStation1) THEN
				xError:=TRUE;
				iStepError:=400;
			END_IF;
		400:	IF xQuitErr THEN
				T_Station.TControl.xQuitError:=T_Station.TControl.xError;
				iStepError:=500;
			END_IF;
		500: IF NOT(T_Station.TControl.xQuitError) THEN
				xSetEnd:=TRUE;
			END_IF;
	END_CASE;
END_IF;
(******************************************************************************************************************************************)
(****************************				              Main Controlling Part                                            *****************************)
(******************************************************************************************************************************************)
IF (xStart OR xStartMainCtr) AND NOT(xSetEnd) AND NOT(xSetError) THEN
	IF NOT (xInitMainCtr) THEN
		iStepPrc:=10;
		xInitMainCtr:=TRUE;
		xStartMainCtr:=TRUE;
		xStart:=FALSE;
		xEnd:=FALSE;
		xSetEndPrc:=FALSE;
		iTmpFunctionNr:=1;
		xAbord:=FALSE;
	END_IF;
	IF xStop AND NOT(xTmpStop) THEN
		xTmpStop:=TRUE;
		iStepStop:=1;
	END_IF;
	IF xTmpStop THEN
		CASE iStepStop OF
		1:	IF NOT(T_Station.TControl.xEnd) THEN
				T_Station.TControl.xStop:=TRUE;
				iStepStop:=10;
			ELSE
				iStepStop:=20;
			END_IF;
		10:	IF NOT(T_Station.TControl.xStop) THEN
				iStepStop:=20;
			END_IF;
		(* Check Active Movement of the Axis *)
		20:	IF NOT(T_Station.TControl.xStart) AND T_Station.TControl.xEnd THEN
				T_Station.TControl.iFunctNr:=18;	(* Check Axis Movement, and stop it if moves *)
				T_Station.TControl.xStart:=TRUE;
				iStepStop:=30;
			END_IF;
		30:	IF NOT(T_Station.TControl.xStart) AND T_Station.TControl.xEnd THEN
				xStartMainPrc:=FALSE;
				xInitStep:=FALSE;
				iStepPrc:=0;
				xSetEnd:=TRUE;
				RETURN;
			END_IF;
		END_CASE;
		RETURN;
	END_IF;
	IF NOT(xStartMainPrc) THEN
		xStartMainPrc:=TRUE;
	END_IF;
END_IF;
(******************************************************************************************************************************************)
(****************************				             Main Procedure Part                                             *****************************)
(******************************************************************************************************************************************)
IF xStartMainPrc AND NOT(xSetEnd) AND NOT(xSetError) THEN
	CASE iStepPrc OF
		(* Check first if the ToolCalibration is available to start it *)
		10:	T_Station.THardware.TAxisToolLeft.T_CtrleSingle.lrAcceleration:=T_NovRAMData.T_Standard.T_TeachINToolLeft.rAcceleration;
			T_Station.THardware.TAxisToolLeft.T_CtrleSingle.lrDecceleration:=T_NovRAMData.T_Standard.T_TeachINToolLeft.rDeceleration;
			T_Station.THardware.TAxisToolCenter.T_CtrleSingle.lrAcceleration:=T_NovRAMData.T_Standard.T_TeachINToolCenter.rAcceleration;
			T_Station.THardware.TAxisToolCenter.T_CtrleSingle.lrDecceleration:=T_NovRAMData.T_Standard.T_TeachINToolCenter.rDeceleration;
			T_Station.THardware.TAxisToolRight.T_CtrleSingle.lrAcceleration:=T_NovRAMData.T_Standard.T_TeachINToolRight.rAcceleration;
			T_Station.THardware.TAxisToolRight.T_CtrleSingle.lrDecceleration:=T_NovRAMData.T_Standard.T_TeachINToolRight.rDeceleration;
			T_Station.THardware.TAxisToolFeeder.T_CtrleSingle.lrAcceleration:=T_NovRAMData.T_Standard.T_TeachINToolFeeder.rAcceleration;
			T_Station.THardware.TAxisToolFeeder.T_CtrleSingle.lrDecceleration:=T_NovRAMData.T_Standard.T_TeachINToolFeeder.rDeceleration;
			T_Station.THardware.TAxisGrindFeeder.T_CtrleSingle.lrAcceleration:=T_NovRAMData.T_Standard.T_TeachINGrindFeeder.rAcceleration;
			T_Station.THardware.TAxisGrindFeeder.T_CtrleSingle.lrDecceleration:=T_NovRAMData.T_Standard.T_TeachINGrindFeeder.rDeceleration;
			(* On the MicroWire it is not possible to start the Reference Procedure *)
			IF NOT(xMicroRodActive) THEN
				xSetError:=TRUE;
				diTmpErrNr:=5;	(* On the MicroWire it is not possible to Referencing *)
				RETURN;
			END_IF;
			xStartMainPrc:=FALSE;
			xInitStep:=FALSE;
			iStepPrc:=20;
		(* Switch First all Axis the power supply on *)
		20:	IF NOT(xInitStep) THEN
				xInitStep:=TRUE;
				T_Station.TControl.iFunctNr:=16;
				T_Station.TControl.xStart:=TRUE;
			END_IF;
			IF NOT(T_Station.TControl.xStart) AND T_Station.TControl.xEnd THEN
				iStepPrc:=30;
				xStartMainPrc:=FALSE;
				xInitStep:=FALSE;
				iTmpStationFunctionNr:=6;
				T_Station.THardware.TAxisToolLeft.T_CtrleSingle.rSetPosition:=0.0;
				T_Station.THardware.TAxisToolCenter.T_CtrleSingle.rSetPosition:=0.0;
				T_Station.THardware.TAxisToolRight.T_CtrleSingle.rSetPosition:=0.0;
				T_Station.THardware.TAxisToolFeeder.T_CtrleSingle.rSetPosition:=0.0;
			END_IF;
		(* Reset the Position of the Axis *)
		30:	IF NOT(xInitStep) THEN
				xInitStep:=TRUE;
				(* 6=ToolLeft, 7=ToolCenter, 8=ToolRight, 9=ToolFeeder *)
				T_Station.TControl.iFunctNr:=iTmpStationFunctionNr;
				T_Station.TControl.xStart:=TRUE;
			END_IF;
			IF NOT(T_Station.TControl.xStart) AND T_Station.TControl.xEnd THEN
				iTmpStationFunctionNr:=iTmpStationFunctionNr + 1;
				xStartMainPrc:=FALSE;
				xInitStep:=FALSE;
				IF (iTmpStationFunctionNr < 10) THEN
					iStepPrc:=30;
				ELSE
					iStepPrc:=40;
				END_IF;
			END_IF;
		(* GrindFeeder Set Absolut to Security Position *)
		40:	IF NOT(xInitStep) THEN
				xInitStep:=TRUE;
				T_Station.TControl.iFunctNr:=4;
				T_Station.TControl.xStart:=TRUE;
				T_Station.THardware.TAxisGrindFeeder.T_CtrleSingle.lrAcceleration:=T_NovRAMData.T_Standard.T_TeachINGrindFeeder.rAcceleration;
				T_Station.THardware.TAxisGrindFeeder.T_CtrleSingle.lrDecceleration:=T_NovRAMData.T_Standard.T_TeachINGrindFeeder.rDeceleration;
				T_Station.THardware.TAxisGrindFeeder.T_CtrleSingle.lrPosition:=	T_NovRAMData.T_ProcessImageData.T_ProcessPara.rToolDiameterProcess +
																			T_NovRAMData.T_ProcessImageData.T_ProcessPara.rSecurityPosGrindFeedProcess;
				T_Station.THardware.TAxisGrindFeeder.T_CtrleSingle.lrVelocity:=T_NovRAMData.T_ProcessImageData.T_ProcessPara.rSpeedBackwardGrindFeed;
			END_IF;
			IF NOT(T_Station.TControl.xStart) AND T_Station.TControl.xEnd THEN
				iStepPrc:=50;
				xStartMainPrc:=FALSE;
				xInitStep:=FALSE;
			END_IF;
		(* Reference the ToolFeeder *)
		50:	IF NOT(xInitStep) THEN
				xStartProcess:=TRUE;
				xInitStep:=TRUE;
				T_Station.TControl.iFunctNr:=1;
				T_Station.TControl.xStart:=TRUE;
			END_IF;
			IF NOT(T_Station.TControl.xStart) AND T_Station.TControl.xEnd THEN
				xStartMainPrc:=FALSE;
				xInitStep:=FALSE;
				iStepPrc:=60;
			END_IF;
		60:	xSetEndPrc:=FALSE;
			xStartMainPrc:=FALSE;
			xInitStep:=FALSE;
			iStepPrc:=0;
			xSetEnd:=TRUE;
	END_CASE;
END_IF;
(******************************************************************************************************************************************)
(****************************				             	Init / Reset Part                                                   *****************************)
(******************************************************************************************************************************************)
IF xSetEnd THEN
	xEnd:=TRUE;
	xInitStep:=FALSE;
	xSetEnd:=FALSE;
	xStop:=FALSE;
	xStartMainPrc:=FALSE;
	xTmpStop:=FALSE;
	xInitMainCtr:=FALSE;
	xStartMainCtr:=FALSE;
	xStart:=FALSE;
	xSetError:=FALSE;
	xQuitErr:=FALSE;
	xError:=FALSE;
	diErrorNr:=0;
	xInitError:=FALSE;
	xFreeze:=FALSE;
	xAbord:=FALSE;
	xTmpAbord:=FALSE;
	xSetEndPrc:=FALSE;
	xStartProcess:=FALSE;
END_IF;
END_FUNCTION_BLOCK

(* POU PRG_PROCESS_LAYER4/FB_PROCESS/FB_PrcAutoGeometry, ST *)
FUNCTION_BLOCK FB_PrcAutoGeometry
VAR_INPUT
	xMicroRodActive: BOOL;				(* choice of the machine MicroWire or MicroRod *)
	xBeckhoffDriveActive: BOOL;			(* choice of the axis Beckhoff or EcoStep *)
	T_NovRAMData:ST_DATA_RETAIN;	(* Novram structure for all Machine parameter *)
END_VAR
VAR_IN_OUT
	xStart : BOOL;							(* start a process *)
	xStop : BOOL;							(* stop a process *)
	xStopCycle : BOOL;					(* stop a process on the end of the cycle *)
	xQuitErr : BOOL;						(* quit an error *)
	xAbord : BOOL;						(* abord a process *)
	T_Station : ST_STATION;				(* data structure of the stationlevel *)
	T_Process : ST_PROCESS;			(* data strucuture of the processlevel *)
	xReset : BOOL;						(* reset the FB *)
	T_ExchgParam:ST_QVIS_EXCHG_PARAM;	(* data structure of the visualisation *)
END_VAR
VAR_OUTPUT
	xEnd : BOOL;							(* Endflag of the process *)
	xError : BOOL;							(* Errorflag of the process *)
	diErrorNr : DINT;						(* Error number of the process *)
END_VAR
VAR
	iStepPrc: INT;
	xInitStep: BOOL;
	xSetError: BOOL;
	xSetEnd: BOOL;
	xStartMainCtr: BOOL;
	xStartMainPrc: BOOL;
	xInitMainCtr: BOOL;
	xFreeze: BOOL;
	xInitError: BOOL;
	iStepError: INT;
	xTmpStop: BOOL;
	xSetTmpError: BOOL;
	xTmpAbord: BOOL;
	diTmpErrNr: DINT;
	xSetEndPrc : BOOL;
	iTmpFunctionNr:INT;
	xStopFctStation1: BOOL;
	iStepStop: INT;
	FBCheckToolGeometryPara: FB_CheckToolGeometryPara;
	iTmpStationFunctionNr: INT;
	xStartProcess: BOOL;
	TONStartTimer: TON;
	tStepTime: TIME;
	TONStartTimer1: TON;
	xDoNotMovePositionOfToolFeeder: BOOL;
	xTmp: BOOL;
	xTmpStopCycle: BOOL;
	xProcessHold: BOOL;
(*08.07.2014: KFS	{	*)
	TONWarmUpBreakTimer: TON;
	TONWarmUpTimer: TON;
	xWarmUpCycle:BOOL;
	xWarmUp:BOOL;
	xWarmUpDone: BOOL;
(*08.07.2014: KFS	}	*)
	TONWaitForTableMovement: TON;
END_VAR
(****************************************************************************************************************************************************)
(***********                                      This Functionblock define the process for the AutoGeometry                                                     ************)
(****************************************************************************************************************************************************)

